LIN {X 0,Y 524.943,Z 315.664,A -85,B 0,C 180,E1 -4750.039,E2 -4750.039} C_VEL
LIN {X 0,Y 524.487,Z 334.734,A -85,B 0,C 180,E1 -4753.056,E2 -4753.056} C_VEL
LIN {X 0,Y 524.293,Z 346.228,A -85,B 0,C 180,E1 -4754.846,E2 -4754.846} C_VEL
LIN {X 0,Y 525.936,Z 357.339,A -85,B 0,C 180,E1 -4755.048,E2 -4755.048} C_VEL
LIN {X 0,Y 525.54,Z 454.207,A -85,B 0,C 180,E1 -4756.393,E2 -4756.393} C_VEL
LIN {X 0,Y 525.313,Z 467.512,A -85,B 0,C 180,E1 -4756.731,E2 -4756.731} C_VEL
LIN {X 0,Y 525.043,Z 480.819,A -85,B 0,C 180,E1 -4757.241,E2 -4757.241} C_VEL
LIN {X 0,Y 524.811,Z 492.313,A -85,B 0,C 180,E1 -4757.845,E2 -4757.845} C_VEL
LIN {X 0,Y 524.527,Z 503.595,A -85,B 0,C 180,E1 -4758.602,E2 -4758.602} C_VEL
LIN {X 0,Y 524.201,Z 514.045,A -85,B 0,C 180,E1 -4759.475,E2 -4759.475} C_VEL
LIN {X 0,Y 523.995,Z 522.59,A -85,B 0,C 180,E1 -4760.349,E2 -4760.349} C_VEL
LIN {X 0,Y 523.801,Z 530.474,A -85,B 0,C 180,E1 -4761.319,E2 -4761.319} C_VEL
LIN {X 0,Y 523.605,Z 538.173,A -85,B 0,C 180,E1 -4762.481,E2 -4762.481} C_VEL
LIN {X 0,Y 523.482,Z 545.27,A -85,B 0,C 180,E1 -4763.835,E2 -4763.835} C_VEL
LIN {X 0,Y 523.383,Z 549.99,A -85,B 0,C 180,E1 -4764.993,E2 -4764.993} C_VEL
LIN {X 0,Y 523.443,Z 553.599,A -85,B 0,C 180,E1 -4766.151,E2 -4766.151} C_VEL
LIN {X 0,Y 523.367,Z 555.458,A -85,B 0,C 180,E1 -4766.922,E2 -4766.922} C_VEL
LIN {X 0,Y 523.334,Z 556.852,A -85,B 0,C 180,E1 -4767.692,E2 -4767.692} C_VEL
LIN {X 0,Y 523.25,Z 558.452,A -85,B 0,C 180,E1 -4769.231,E2 -4769.231} C_VEL
LIN {X 0,Y 523.247,Z 558.668,A -85,B 0,C 180,E1 -4770.001,E2 -4770.001} C_VEL
LIN {X 0,Y 523.274,Z 557.844,A -85,B 0,C 180,E1 -4771.54,E2 -4771.54} C_VEL
LIN {X 0,Y 523.334,Z 556.851,A -85,B 0,C 180,E1 -4772.309,E2 -4772.309} C_VEL
LIN {X 0,Y 523.368,Z 555.456,A -85,B 0,C 180,E1 -4773.08,E2 -4773.08} C_VEL
LIN {X 0,Y 523.424,Z 552.521,A -85,B 0,C 180,E1 -4774.236,E2 -4774.236} C_VEL
LIN {X 0,Y 523.461,Z 548.548,A -85,B 0,C 180,E1 -4775.393,E2 -4775.393} C_VEL
LIN {X 0,Y 523.515,Z 542.453,A -85,B 0,C 180,E1 -4776.743,E2 -4776.743} C_VEL
LIN {X 0,Y 523.667,Z 535.757,A -85,B 0,C 180,E1 -4777.907,E2 -4777.907} C_VEL
LIN {X 0,Y 523.88,Z 527.47,A -85,B 0,C 180,E1 -4779.07,E2 -4779.07} C_VEL
LIN {X 0,Y 524.072,Z 518.975,A -85,B 0,C 180,E1 -4780.04,E2 -4780.04} C_VEL
LIN {X 0,Y 524.352,Z 508.478,A -85,B 0,C 180,E1 -4781.011,E2 -4781.011} C_VEL
LIN {X 0,Y 524.634,Z 498.216,A -85,B 0,C 180,E1 -4781.78,E2 -4781.78} C_VEL
LIN {X 0,Y 524.943,Z 486.709,A -85,B 0,C 180,E1 -4782.468,E2 -4782.468} C_VEL
LIN {X 0,Y 525.177,Z 475.02,A -85,B 0,C 180,E1 -4783.003,E2 -4783.003} C_VEL
LIN {X 0,Y 525.393,Z 461.551,A -85,B 0,C 180,E1 -4783.44,E2 -4783.44} C_VEL
LIN {X 0,Y 525.574,Z 448.203,A -85,B 0,C 180,E1 -4783.706,E2 -4783.706} C_VEL
LIN {X 0,Y 525.813,Z 355.915,A -85,B 0,C 180,E1 -4784.975,E2 -4784.975} C_VEL
LIN {X 0,Y 524.25,Z 345.993,A -85,B 0,C 180,E1 -4785.173,E2 -4785.173} C_VEL
LIN {X 0,Y 524.694,Z 325.97,A -85,B 0,C 180,E1 -4788.307,E2 -4788.307} C_VEL
LIN {X 0,Y 525.128,Z 306.537,A -85,B 0,C 180,E1 -4791.389,E2 -4791.389} C_VEL
LIN {X 0,Y 525.254,Z 297.571,A -85,B 0,C 180,E1 -4792.832,E2 -4792.832} C_VEL
LIN {X 0,Y 523.921,Z 290.224,A -85,B 0,C 180,E1 -4794.108,E2 -4794.108} C_VEL
LIN {X 0,Y 523.948,Z 290.22,A -85,B 0,C 180,E1 -4797.134,E2 -4797.134} C_VEL
LIN {X 0,Y 523.939,Z 290.226,A -85,B 0,C 180,E1 -4799.756,E2 -4799.756} C_VEL
LIN {X 0,Y 523.936,Z 290.22,A -85,B 0,C 180,E1 -4802.45,E2 -4802.45} C_VEL
LIN {X 0,Y 523.92,Z 290.22,A -85,B 0,C 180,E1 -4805.227,E2 -4805.227} C_VEL
LIN {X 0,Y 523.915,Z 290.227,A -85,B 0,C 180,E1 -4808.102,E2 -4808.102} C_VEL
LIN {X 0,Y 523.955,Z 290.213,A -85,B 0,C 180,E1 -4811.31,E2 -4811.31} C_VEL
LIN {X 0,Y 523.939,Z 290.22,A -85,B 0,C 180,E1 -4814.689,E2 -4814.689} C_VEL
LIN {X 0,Y 523.944,Z 290.217,A -85,B 0,C 180,E1 -4817.88,E2 -4817.88} C_VEL
LIN {X 0,Y 523.92,Z 290.221,A -85,B 0,C 180,E1 -4820.915,E2 -4820.915} C_VEL
LIN {X 0,Y 523.896,Z 290.22,A -85,B 0,C 180,E1 -4823.825,E2 -4823.825} C_VEL
LIN {X 0,Y 523.942,Z 290.222,A -85,B 0,C 180,E1 -4826.636,E2 -4826.636} C_VEL
LIN {X 0,Y 523.95,Z 290.217,A -85,B 0,C 180,E1 -4829.355,E2 -4829.355} C_VEL
LIN {X 0,Y 523.947,Z 290.214,A -85,B 0,C 180,E1 -4832.288,E2 -4832.288} C_VEL
LIN {X 0,Y 523.907,Z 290.224,A -85,B 0,C 180,E1 -4835.427,E2 -4835.427} C_VEL
LIN {X 0,Y 523.938,Z 290.216,A -85,B 0,C 180,E1 -4837.939,E2 -4837.939} C_VEL
LIN {X 0,Y 523.974,Z 290.21,A -85,B 0,C 180,E1 -4840.408,E2 -4840.408} C_VEL
LIN {X 0,Y 523.955,Z 290.214,A -85,B 0,C 180,E1 -4842.837,E2 -4842.837} C_VEL
LIN {X 0,Y 523.977,Z 290.215,A -85,B 0,C 180,E1 -4845.236,E2 -4845.236} C_VEL
LIN {X 0,Y 524.014,Z 290.205,A -85,B 0,C 180,E1 -4848.394,E2 -4848.394} C_VEL
LIN {X 0,Y 523.986,Z 290.213,A -85,B 0,C 180,E1 -4851.516,E2 -4851.516} C_VEL
LIN {X 0,Y 524.033,Z 290.212,A -85,B 0,C 180,E1 -4853.841,E2 -4853.841} C_VEL
LIN {X 0,Y 524.033,Z 290.201,A -85,B 0,C 180,E1 -4856.925,E2 -4856.925} C_VEL
LIN {X 0,Y 524.116,Z 290.2,A -85,B 0,C 180,E1 -4860,E2 -4860} C_VEL
LIN {X 0,Y 524.038,Z 290.202,A -85,B 0,C 180,E1 -4863.075,E2 -4863.075} C_VEL
LIN {X 0,Y 524.028,Z 290.209,A -85,B 0,C 180,E1 -4866.159,E2 -4866.159} C_VEL
LIN {X 0,Y 523.987,Z 290.207,A -85,B 0,C 180,E1 -4869.262,E2 -4869.262} C_VEL
LIN {X 0,Y 524.001,Z 290.208,A -85,B 0,C 180,E1 -4871.738,E2 -4871.738} C_VEL
LIN {X 0,Y 523.995,Z 290.212,A -85,B 0,C 180,E1 -4875.052,E2 -4875.052} C_VEL
LIN {X 0,Y 523.948,Z 290.212,A -85,B 0,C 180,E1 -4877.97,E2 -4877.97} C_VEL
LIN {X 0,Y 523.973,Z 290.214,A -85,B 0,C 180,E1 -4880.41,E2 -4880.41} C_VEL
LIN {X 0,Y 523.911,Z 290.226,A -85,B 0,C 180,E1 -4882.894,E2 -4882.894} C_VEL
LIN {X 0,Y 523.931,Z 290.219,A -85,B 0,C 180,E1 -4885.42,E2 -4885.42} C_VEL
LIN {X 0,Y 523.919,Z 290.216,A -85,B 0,C 180,E1 -4888.002,E2 -4888.002} C_VEL
LIN {X 0,Y 523.941,Z 290.218,A -85,B 0,C 180,E1 -4890.854,E2 -4890.854} C_VEL
LIN {X 0,Y 523.932,Z 290.219,A -85,B 0,C 180,E1 -4893.73,E2 -4893.73} C_VEL
LIN {X 0,Y 523.901,Z 290.22,A -85,B 0,C 180,E1 -4896.401,E2 -4896.401} C_VEL
LIN {X 0,Y 523.923,Z 290.22,A -85,B 0,C 180,E1 -4899.085,E2 -4899.085} C_VEL
LIN {X 0,Y 523.943,Z 290.219,A -85,B 0,C 180,E1 -4902.12,E2 -4902.12} C_VEL
LIN {X 0,Y 523.941,Z 290.218,A -85,B 0,C 180,E1 -4905.311,E2 -4905.311} C_VEL
LIN {X 0,Y 523.89,Z 290.223,A -85,B 0,C 180,E1 -4906.901,E2 -4906.901} C_VEL
LIN {X 0,Y 523.213,Z 290.312,A -85,B 0,C 180,E1 -4907.543,E2 -4907.543} C_VEL
LIN {X 0,Y 520.366,Z 290.672,A -85,B 0,C 180,E1 -4908.584,E2 -4908.584} C_VEL
LIN {X 0,Y 517.968,Z 290.974,A -85,B 0,C 180,E1 -4909.423,E2 -4909.423} C_VEL
LIN {X 0,Y 516.943,Z 291.098,A -85,B 0,C 180,E1 -4910.071,E2 -4910.071} C_VEL
LIN {X 0,Y 516.861,Z 291.105,A -85,B 0,C 180,E1 -4910.29,E2 -4910.29} C_VEL
LIN {X 0,Y 516.848,Z 291.102,A -85,B 0,C 180,E1 -4913.251,E2 -4913.251} C_VEL
LIN {X 0,Y 516.884,Z 291.102,A -85,B 0,C 180,E1 -4916.119,E2 -4916.119} C_VEL
LIN {X 0,Y 516.96,Z 291.244,A -85,B 0,C 180,E1 -4918.668,E2 -4918.668} C_VEL
LIN {X 0,Y 517.503,Z 296.303,A -85,B 0,C 180,E1 -4919.61,E2 -4919.61} C_VEL
LIN {X 0,Y 517.294,Z 312.213,A -85,B 0,C 180,E1 -4922.488,E2 -4922.488} C_VEL
LIN {X 0,Y 517.239,Z 318.815,A -85,B 0,C 180,E1 -4923.684,E2 -4923.684} C_VEL
LIN {X 0,Y 519.136,Z 329.983,A -85,B 0,C 180,E1 -4923.905,E2 -4923.905} C_VEL
LIN {X 0,Y 518.627,Z 426.694,A -85,B 0,C 180,E1 -4925.272,E2 -4925.272} C_VEL
LIN {X 0,Y 518.413,Z 439.775,A -85,B 0,C 180,E1 -4925.619,E2 -4925.619} C_VEL
LIN {X 0,Y 518.18,Z 451.968,A -85,B 0,C 180,E1 -4926.097,E2 -4926.097} C_VEL
LIN {X 0,Y 517.912,Z 463.726,A -85,B 0,C 180,E1 -4926.72,E2 -4926.72} C_VEL
LIN {X 0,Y 517.595,Z 475.325,A -85,B 0,C 180,E1 -4927.515,E2 -4927.515} C_VEL
LIN {X 0,Y 517.267,Z 485.379,A -85,B 0,C 180,E1 -4928.374,E2 -4928.374} C_VEL
LIN {X 0,Y 517.028,Z 494.258,A -85,B 0,C 180,E1 -4929.303,E2 -4929.303} C_VEL
LIN {X 0,Y 516.78,Z 502.321,A -85,B 0,C 180,E1 -4930.33,E2 -4930.33} C_VEL
LIN {X 0,Y 516.573,Z 510.116,A -85,B 0,C 180,E1 -4931.559,E2 -4931.559} C_VEL
LIN {X 0,Y 516.487,Z 515.377,A -85,B 0,C 180,E1 -4932.58,E2 -4932.58} C_VEL
LIN {X 0,Y 516.352,Z 520.412,A -85,B 0,C 180,E1 -4933.798,E2 -4933.798} C_VEL
LIN {X 0,Y 516.305,Z 524.542,A -85,B 0,C 180,E1 -4935.121,E2 -4935.121} C_VEL
LIN {X 0,Y 516.198,Z 527.693,A -85,B 0,C 180,E1 -4936.617,E2 -4936.617} C_VEL
LIN {X 0,Y 516.249,Z 529.366,A -85,B 0,C 180,E1 -4938.217,E2 -4938.217} C_VEL
LIN {X 0,Y 516.259,Z 529.606,A -85,B 0,C 180,E1 -4939.013,E2 -4939.013} C_VEL
LIN {X 0,Y 516.241,Z 529.405,A -85,B 0,C 180,E1 -4939.806,E2 -4939.806} C_VEL
LIN {X 0,Y 516.215,Z 527.808,A -85,B 0,C 180,E1 -4941.387,E2 -4941.387} C_VEL
LIN {X 0,Y 516.273,Z 526.41,A -85,B 0,C 180,E1 -4942.176,E2 -4942.176} C_VEL
LIN {X 0,Y 516.318,Z 522.893,A -85,B 0,C 180,E1 -4943.548,E2 -4943.548} C_VEL
LIN {X 0,Y 516.383,Z 517.948,A -85,B 0,C 180,E1 -4944.924,E2 -4944.924} C_VEL
LIN {X 0,Y 516.536,Z 512.457,A -85,B 0,C 180,E1 -4946.099,E2 -4946.099} C_VEL
LIN {X 0,Y 516.647,Z 505.638,A -85,B 0,C 180,E1 -4947.271,E2 -4947.271} C_VEL
LIN {X 0,Y 516.968,Z 497.099,A -85,B 0,C 180,E1 -4948.441,E2 -4948.441} C_VEL
LIN {X 0,Y 517.173,Z 488.4,A -85,B 0,C 180,E1 -4949.415,E2 -4949.415} C_VEL
LIN {X 0,Y 517.449,Z 477.72,A -85,B 0,C 180,E1 -4950.389,E2 -4950.389} C_VEL
LIN {X 0,Y 517.843,Z 466.961,A -85,B 0,C 180,E1 -4951.166,E2 -4951.166} C_VEL
LIN {X 0,Y 518.127,Z 454.986,A -85,B 0,C 180,E1 -4951.846,E2 -4951.846} C_VEL
LIN {X 0,Y 518.343,Z 442.502,A -85,B 0,C 180,E1 -4952.379,E2 -4952.379} C_VEL
LIN {X 0,Y 518.557,Z 430.182,A -85,B 0,C 180,E1 -4952.743,E2 -4952.743} C_VEL
LIN {X 0,Y 518.683,Z 414.633,A -85,B 0,C 180,E1 -4953.009,E2 -4953.009} C_VEL
LIN {X 0,Y 519.008,Z 328.91,A -85,B 0,C 180,E1 -4954.204,E2 -4954.204} C_VEL
LIN {X 0,Y 517.196,Z 318.905,A -85,B 0,C 180,E1 -4954.408,E2 -4954.408} C_VEL
LIN {X 0,Y 517.583,Z 301.777,A -85,B 0,C 180,E1 -4957.59,E2 -4957.59} C_VEL
LIN {X 0,Y 517.593,Z 295.417,A -85,B 0,C 180,E1 -4958.786,E2 -4958.786} C_VEL
LIN {X 0,Y 516.941,Z 291.096,A -85,B 0,C 180,E1 -4959.636,E2 -4959.636} C_VEL
LIN {X 0,Y 516.907,Z 291.095,A -85,B 0,C 180,E1 -4962.564,E2 -4962.564} C_VEL
LIN {X 0,Y 516.946,Z 291.086,A -85,B 0,C 180,E1 -4965.145,E2 -4965.145} C_VEL
LIN {X 0,Y 516.877,Z 291.101,A -85,B 0,C 180,E1 -4968.223,E2 -4968.223} C_VEL
LIN {X 0,Y 516.901,Z 291.093,A -85,B 0,C 180,E1 -4970.701,E2 -4970.701} C_VEL
LIN {X 0,Y 516.857,Z 291.097,A -85,B 0,C 180,E1 -4973.223,E2 -4973.223} C_VEL
LIN {X 0,Y 516.868,Z 291.104,A -85,B 0,C 180,E1 -4976.178,E2 -4976.178} C_VEL
LIN {X 0,Y 516.902,Z 291.091,A -85,B 0,C 180,E1 -4979.305,E2 -4979.305} C_VEL
LIN {X 0,Y 516.89,Z 291.102,A -85,B 0,C 180,E1 -4982.541,E2 -4982.541} C_VEL
LIN {X 0,Y 516.851,Z 291.098,A -85,B 0,C 180,E1 -4985.326,E2 -4985.326} C_VEL
LIN {X 0,Y 516.868,Z 291.106,A -85,B 0,C 180,E1 -4988.716,E2 -4988.716} C_VEL
LIN {X 0,Y 516.84,Z 291.099,A -85,B 0,C 180,E1 -4991.781,E2 -4991.781} C_VEL
LIN {X 0,Y 516.891,Z 291.101,A -85,B 0,C 180,E1 -4995.006,E2 -4995.006} C_VEL
LIN {X 0,Y 516.845,Z 291.1,A -85,B 0,C 180,E1 -4998.406,E2 -4998.406} C_VEL
LIN {X 0,Y 516.865,Z 291.103,A -85,B 0,C 180,E1 -5001.282,E2 -5001.282} C_VEL
LIN {X 0,Y 516.844,Z 291.101,A -85,B 0,C 180,E1 -5004.672,E2 -5004.672} C_VEL
LIN {X 0,Y 516.856,Z 291.104,A -85,B 0,C 180,E1 -5007.462,E2 -5007.462} C_VEL
LIN {X 0,Y 516.836,Z 291.1,A -85,B 0,C 180,E1 -5010.489,E2 -5010.489} C_VEL
LIN {X 0,Y 516.818,Z 291.109,A -85,B 0,C 180,E1 -5013.336,E2 -5013.336} C_VEL
LIN {X 0,Y 516.86,Z 291.101,A -85,B 0,C 180,E1 -5015.925,E2 -5015.925} C_VEL
LIN {X 0,Y 516.869,Z 291.096,A -85,B 0,C 180,E1 -5018.461,E2 -5018.461} C_VEL
LIN {X 0,Y 516.861,Z 291.097,A -85,B 0,C 180,E1 -5020.953,E2 -5020.953} C_VEL
LIN {X 0,Y 516.818,Z 291.106,A -85,B 0,C 180,E1 -5023.407,E2 -5023.407} C_VEL
LIN {X 0,Y 516.844,Z 291.108,A -85,B 0,C 180,E1 -5025.832,E2 -5025.832} C_VEL
LIN {X 0,Y 516.916,Z 291.095,A -85,B 0,C 180,E1 -5028.232,E2 -5028.232} C_VEL
LIN {X 0,Y 516.909,Z 291.092,A -85,B 0,C 180,E1 -5031.398,E2 -5031.398} C_VEL
LIN {X 0,Y 516.97,Z 291.087,A -85,B 0,C 180,E1 -5034.539,E2 -5034.539} C_VEL
LIN {X 0,Y 517.062,Z 291.073,A -85,B 0,C 180,E1 -5037.663,E2 -5037.663} C_VEL
LIN {X 0,Y 517.079,Z 291.073,A -85,B 0,C 180,E1 -5040.779,E2 -5040.779} C_VEL
LIN {X 0,Y 516.957,Z 291.085,A -85,B 0,C 180,E1 -5043.117,E2 -5043.117} C_VEL
LIN {X 0,Y 516.972,Z 291.088,A -85,B 0,C 180,E1 -5046.244,E2 -5046.244} C_VEL
LIN {X 0,Y 516.922,Z 291.089,A -85,B 0,C 180,E1 -5049.39,E2 -5049.39} C_VEL
LIN {X 0,Y 516.943,Z 291.086,A -85,B 0,C 180,E1 -5051.807,E2 -5051.807} C_VEL
LIN {X 0,Y 516.927,Z 291.093,A -85,B 0,C 180,E1 -5055.143,E2 -5055.143} C_VEL
LIN {X 0,Y 516.902,Z 291.092,A -85,B 0,C 180,E1 -5058.223,E2 -5058.223} C_VEL
LIN {X 0,Y 516.895,Z 291.097,A -85,B 0,C 180,E1 -5060.702,E2 -5060.702} C_VEL
LIN {X 0,Y 516.876,Z 291.095,A -85,B 0,C 180,E1 -5064.074,E2 -5064.074} C_VEL
LIN {X 0,Y 516.894,Z 291.095,A -85,B 0,C 180,E1 -5066.66,E2 -5066.66} C_VEL
LIN {X 0,Y 516.9,Z 291.097,A -85,B 0,C 180,E1 -5069.524,E2 -5069.524} C_VEL
LIN {X 0,Y 516.888,Z 291.093,A -85,B 0,C 180,E1 -5072.544,E2 -5072.544} C_VEL
LIN {X 0,Y 516.856,Z 291.105,A -85,B 0,C 180,E1 -5075.33,E2 -5075.33} C_VEL
LIN {X 0,Y 516.871,Z 291.099,A -85,B 0,C 180,E1 -5077.943,E2 -5077.943} C_VEL
LIN {X 0,Y 516.875,Z 291.095,A -85,B 0,C 180,E1 -5080.743,E2 -5080.743} C_VEL
LIN {X 0,Y 516.875,Z 291.102,A -85,B 0,C 180,E1 -5083.904,E2 -5083.904} C_VEL
LIN {X 0,Y 516.876,Z 291.1,A -85,B 0,C 180,E1 -5086.108,E2 -5086.108} C_VEL
LIN {X 0,Y 516.877,Z 291.096,A -85,B 0,C 180,E1 -5089.259,E2 -5089.259} C_VEL
LIN {X 0,Y 516.857,Z 291.102,A -85,B 0,C 180,E1 -5092.275,E2 -5092.275} C_VEL
LIN {X 0,Y 516.878,Z 291.094,A -85,B 0,C 180,E1 -5095.176,E2 -5095.176} C_VEL
LIN {X 0,Y 516.871,Z 291.102,A -85,B 0,C 180,E1 -5097.976,E2 -5097.976} C_VEL
LIN {X 0,Y 516.918,Z 291.094,A -85,B 0,C 180,E1 -5100.696,E2 -5100.696} C_VEL
LIN {X 0,Y 516.9,Z 291.096,A -85,B 0,C 180,E1 -5103.814,E2 -5103.814} C_VEL
LIN {X 0,Y 516.91,Z 291.275,A -85,B 0,C 180,E1 -5105.728,E2 -5105.728} C_VEL
LIN {X 0,Y 518.388,Z 299.806,A -85,B 0,C 180,E1 -5107.206,E2 -5107.206} C_VEL
LIN {X 0,Y 517.915,Z 318.019,A -85,B 0,C 180,E1 -5110.17,E2 -5110.17} C_VEL
LIN {X 0,Y 517.456,Z 335.805,A -85,B 0,C 180,E1 -5113.022,E2 -5113.022} C_VEL
LIN {X 0,Y 517.281,Z 346.006,A -85,B 0,C 180,E1 -5114.635,E2 -5114.635} C_VEL
LIN {X 0,Y 519.07,Z 358.553,A -85,B 0,C 180,E1 -5114.865,E2 -5114.865} C_VEL
LIN {X 0,Y 518.653,Z 453.984,A -85,B 0,C 180,E1 -5116.208,E2 -5116.208} C_VEL
LIN {X 0,Y 518.387,Z 467.297,A -85,B 0,C 180,E1 -5116.551,E2 -5116.551} C_VEL
LIN {X 0,Y 518.134,Z 480.61,A -85,B 0,C 180,E1 -5117.068,E2 -5117.068} C_VEL
LIN {X 0,Y 517.823,Z 493.124,A -85,B 0,C 180,E1 -5117.742,E2 -5117.742} C_VEL
LIN {X 0,Y 517.51,Z 504.686,A -85,B 0,C 180,E1 -5118.545,E2 -5118.545} C_VEL
LIN {X 0,Y 517.154,Z 514.888,A -85,B 0,C 180,E1 -5119.429,E2 -5119.429} C_VEL
LIN {X 0,Y 516.931,Z 524.07,A -85,B 0,C 180,E1 -5120.414,E2 -5120.414} C_VEL
LIN {X 0,Y 516.661,Z 533.013,A -85,B 0,C 180,E1 -5121.592,E2 -5121.592} C_VEL
LIN {X 0,Y 516.508,Z 540.213,A -85,B 0,C 180,E1 -5122.77,E2 -5122.77} C_VEL
LIN {X 0,Y 516.417,Z 546.769,A -85,B 0,C 180,E1 -5124.142,E2 -5124.142} C_VEL
LIN {X 0,Y 516.269,Z 551.103,A -85,B 0,C 180,E1 -5125.316,E2 -5125.316} C_VEL
LIN {X 0,Y 516.352,Z 553.401,A -85,B 0,C 180,E1 -5126.098,E2 -5126.098} C_VEL
LIN {X 0,Y 516.282,Z 555.26,A -85,B 0,C 180,E1 -5126.879,E2 -5126.879} C_VEL
LIN {X 0,Y 516.26,Z 556.654,A -85,B 0,C 180,E1 -5127.66,E2 -5127.66} C_VEL
LIN {X 0,Y 516.16,Z 558.254,A -85,B 0,C 180,E1 -5129.22,E2 -5129.22} C_VEL
LIN {X 0,Y 516.155,Z 558.469,A -85,B 0,C 180,E1 -5130.001,E2 -5130.001} C_VEL
LIN {X 0,Y 516.191,Z 557.646,A -85,B 0,C 180,E1 -5131.561,E2 -5131.561} C_VEL
LIN {X 0,Y 516.26,Z 556.652,A -85,B 0,C 180,E1 -5132.341,E2 -5132.341} C_VEL
LIN {X 0,Y 516.283,Z 555.256,A -85,B 0,C 180,E1 -5133.122,E2 -5133.122} C_VEL
LIN {X 0,Y 516.312,Z 552.32,A -85,B 0,C 180,E1 -5134.294,E2 -5134.294} C_VEL
LIN {X 0,Y 516.375,Z 548.346,A -85,B 0,C 180,E1 -5135.467,E2 -5135.467} C_VEL
LIN {X 0,Y 516.422,Z 543.132,A -85,B 0,C 180,E1 -5136.664,E2 -5136.664} C_VEL
LIN {X 0,Y 516.581,Z 536.79,A -85,B 0,C 180,E1 -5137.82,E2 -5137.82} C_VEL
LIN {X 0,Y 516.785,Z 528.756,A -85,B 0,C 180,E1 -5138.998,E2 -5138.998} C_VEL
LIN {X 0,Y 517.018,Z 520.569,A -85,B 0,C 180,E1 -5139.981,E2 -5139.981} C_VEL
LIN {X 0,Y 517.326,Z 510.586,A -85,B 0,C 180,E1 -5140.965,E2 -5140.965} C_VEL
LIN {X 0,Y 517.628,Z 500.738,A -85,B 0,C 180,E1 -5141.752,E2 -5141.752} C_VEL
LIN {X 0,Y 517.916,Z 489.603,A -85,B 0,C 180,E1 -5142.465,E2 -5142.465} C_VEL
LIN {X 0,Y 518.177,Z 477.153,A -85,B 0,C 180,E1 -5143.082,E2 -5143.082} C_VEL
LIN {X 0,Y 518.424,Z 464.071,A -85,B 0,C 180,E1 -5143.549,E2 -5143.549} C_VEL
LIN {X 0,Y 518.65,Z 451.001,A -85,B 0,C 180,E1 -5143.843,E2 -5143.843} C_VEL
LIN {X 0,Y 518.987,Z 356.904,A -85,B 0,C 180,E1 -5145.16,E2 -5145.16} C_VEL
LIN {X 0,Y 517.241,Z 345.723,A -85,B 0,C 180,E1 -5145.393,E2 -5145.393} C_VEL
LIN {X 0,Y 517.691,Z 326.778,A -85,B 0,C 180,E1 -5148.399,E2 -5148.399} C_VEL
LIN {X 0,Y 518.168,Z 307.605,A -85,B 0,C 180,E1 -5151.482,E2 -5151.482} C_VEL
LIN {X 0,Y 518.305,Z 298.878,A -85,B 0,C 180,E1 -5152.908,E2 -5152.908} C_VEL
LIN {X 0,Y 516.914,Z 291.097,A -85,B 0,C 180,E1 -5154.273,E2 -5154.273} C_VEL
LIN {X 0,Y 516.925,Z 291.1,A -85,B 0,C 180,E1 -5157.533,E2 -5157.533} C_VEL
LIN {X 0,Y 516.889,Z 291.102,A -85,B 0,C 180,E1 -5160.204,E2 -5160.204} C_VEL
LIN {X 0,Y 516.897,Z 291.095,A -85,B 0,C 180,E1 -5162.947,E2 -5162.947} C_VEL
LIN {X 0,Y 516.87,Z 291.104,A -85,B 0,C 180,E1 -5165.781,E2 -5165.781} C_VEL
LIN {X 0,Y 516.879,Z 291.097,A -85,B 0,C 180,E1 -5168.716,E2 -5168.716} C_VEL
LIN {X 0,Y 516.908,Z 291.094,A -85,B 0,C 180,E1 -5171.776,E2 -5171.776} C_VEL
LIN {X 0,Y 516.897,Z 291.094,A -85,B 0,C 180,E1 -5175.007,E2 -5175.007} C_VEL
LIN {X 0,Y 516.911,Z 291.1,A -85,B 0,C 180,E1 -5178.399,E2 -5178.399} C_VEL
LIN {X 0,Y 516.88,Z 291.094,A -85,B 0,C 180,E1 -5181.284,E2 -5181.284} C_VEL
LIN {X 0,Y 516.869,Z 291.098,A -85,B 0,C 180,E1 -5184.219,E2 -5184.219} C_VEL
LIN {X 0,Y 516.896,Z 291.097,A -85,B 0,C 180,E1 -5187.053,E2 -5187.053} C_VEL
LIN {X 0,Y 516.887,Z 291.094,A -85,B 0,C 180,E1 -5189.796,E2 -5189.796} C_VEL
LIN {X 0,Y 516.9,Z 291.093,A -85,B 0,C 180,E1 -5192.466,E2 -5192.466} C_VEL
LIN {X 0,Y 516.849,Z 291.106,A -85,B 0,C 180,E1 -5195.069,E2 -5195.069} C_VEL
LIN {X 0,Y 516.87,Z 291.099,A -85,B 0,C 180,E1 -5197.622,E2 -5197.622} C_VEL
LIN {X 0,Y 516.932,Z 291.088,A -85,B 0,C 180,E1 -5200.13,E2 -5200.13} C_VEL
LIN {X 0,Y 516.906,Z 291.09,A -85,B 0,C 180,E1 -5202.595,E2 -5202.595} C_VEL
LIN {X 0,Y 516.943,Z 291.088,A -85,B 0,C 180,E1 -5205.03,E2 -5205.03} C_VEL
LIN {X 0,Y 516.967,Z 291.084,A -85,B 0,C 180,E1 -5208.234,E2 -5208.234} C_VEL
LIN {X 0,Y 516.954,Z 291.088,A -85,B 0,C 180,E1 -5211.4,E2 -5211.4} C_VEL
LIN {X 0,Y 516.999,Z 291.086,A -85,B 0,C 180,E1 -5213.757,E2 -5213.757} C_VEL
LIN {X 0,Y 516.975,Z 291.08,A -85,B 0,C 180,E1 -5216.883,E2 -5216.883} C_VEL
LIN {X 0,Y 517.091,Z 291.067,A -85,B 0,C 180,E1 -5219.221,E2 -5219.221} C_VEL
LIN {X 0,Y 517.08,Z 291.076,A -85,B 0,C 180,E1 -5222.337,E2 -5222.337} C_VEL
LIN {X 0,Y 517.021,Z 291.074,A -85,B 0,C 180,E1 -5225.46,E2 -5225.46} C_VEL
LIN {X 0,Y 516.964,Z 291.088,A -85,B 0,C 180,E1 -5228.601,E2 -5228.601} C_VEL
LIN {X 0,Y 516.953,Z 291.086,A -85,B 0,C 180,E1 -5231.807,E2 -5231.807} C_VEL
LIN {X 0,Y 516.946,Z 291.089,A -85,B 0,C 180,E1 -5235.147,E2 -5235.147} C_VEL
LIN {X 0,Y 516.917,Z 291.089,A -85,B 0,C 180,E1 -5238.223,E2 -5238.223} C_VEL
LIN {X 0,Y 516.914,Z 291.097,A -85,B 0,C 180,E1 -5240.702,E2 -5240.702} C_VEL
LIN {X 0,Y 516.89,Z 291.092,A -85,B 0,C 180,E1 -5244.073,E2 -5244.073} C_VEL
LIN {X 0,Y 516.9,Z 291.094,A -85,B 0,C 180,E1 -5246.66,E2 -5246.66} C_VEL
LIN {X 0,Y 516.911,Z 291.095,A -85,B 0,C 180,E1 -5249.523,E2 -5249.523} C_VEL
LIN {X 0,Y 516.896,Z 291.092,A -85,B 0,C 180,E1 -5252.543,E2 -5252.543} C_VEL
LIN {X 0,Y 516.867,Z 291.103,A -85,B 0,C 180,E1 -5255.329,E2 -5255.329} C_VEL
LIN {X 0,Y 516.881,Z 291.099,A -85,B 0,C 180,E1 -5257.943,E2 -5257.943} C_VEL
LIN {X 0,Y 516.874,Z 291.096,A -85,B 0,C 180,E1 -5260.743,E2 -5260.743} C_VEL
LIN {X 0,Y 516.884,Z 291.102,A -85,B 0,C 180,E1 -5263.893,E2 -5263.893} C_VEL
LIN {X 0,Y 516.843,Z 291.101,A -85,B 0,C 180,E1 -5266.902,E2 -5266.902} C_VEL
LIN {X 0,Y 516.864,Z 291.102,A -85,B 0,C 180,E1 -5269.593,E2 -5269.593} C_VEL
LIN {X 0,Y 516.861,Z 291.105,A -85,B 0,C 180,E1 -5270.29,E2 -5270.29} C_VEL
LIN {X 0,Y 516.2,Z 291.183,A -85,B 0,C 180,E1 -5270.941,E2 -5270.941} C_VEL
LIN {X 0,Y 513.349,Z 291.543,A -85,B 0,C 180,E1 -5271.996,E2 -5271.996} C_VEL
LIN {X 0,Y 510.932,Z 291.844,A -85,B 0,C 180,E1 -5272.847,E2 -5272.847} C_VEL
LIN {X 0,Y 509.891,Z 291.971,A -85,B 0,C 180,E1 -5273.503,E2 -5273.503} C_VEL
LIN {X 0,Y 509.804,Z 291.982,A -85,B 0,C 180,E1 -5273.726,E2 -5273.726} C_VEL
LIN {X 0,Y 509.844,Z 291.98,A -85,B 0,C 180,E1 -5276.538,E2 -5276.538} C_VEL
LIN {X 0,Y 509.887,Z 292.074,A -85,B 0,C 180,E1 -5278.525,E2 -5278.525} C_VEL
LIN {X 0,Y 510.514,Z 297.753,A -85,B 0,C 180,E1 -5279.597,E2 -5279.597} C_VEL
LIN {X 0,Y 510.296,Z 313.783,A -85,B 0,C 180,E1 -5282.524,E2 -5282.524} C_VEL
LIN {X 0,Y 510.289,Z 319.229,A -85,B 0,C 180,E1 -5283.478,E2 -5283.478} C_VEL
LIN {X 0,Y 512.298,Z 331.341,A -85,B 0,C 180,E1 -5283.714,E2 -5283.714} C_VEL
LIN {X 0,Y 511.745,Z 426.106,A -85,B 0,C 180,E1 -5285.066,E2 -5285.066} C_VEL
LIN {X 0,Y 511.517,Z 439.542,A -85,B 0,C 180,E1 -5285.421,E2 -5285.421} C_VEL
LIN {X 0,Y 511.286,Z 452.079,A -85,B 0,C 180,E1 -5285.916,E2 -5285.916} C_VEL
LIN {X 0,Y 510.952,Z 464.688,A -85,B 0,C 180,E1 -5286.599,E2 -5286.599} C_VEL
LIN {X 0,Y 510.602,Z 476.585,A -85,B 0,C 180,E1 -5287.438,E2 -5287.438} C_VEL
LIN {X 0,Y 510.269,Z 487.146,A -85,B 0,C 180,E1 -5288.381,E2 -5288.381} C_VEL
LIN {X 0,Y 509.984,Z 495.942,A -85,B 0,C 180,E1 -5289.349,E2 -5289.349} C_VEL
LIN {X 0,Y 509.712,Z 504.253,A -85,B 0,C 180,E1 -5290.466,E2 -5290.466} C_VEL
LIN {X 0,Y 509.501,Z 511.63,A -85,B 0,C 180,E1 -5291.691,E2 -5291.691} C_VEL
LIN {X 0,Y 509.405,Z 516.726,A -85,B 0,C 180,E1 -5292.745,E2 -5292.745} C_VEL
LIN {X 0,Y 509.277,Z 521.514,A -85,B 0,C 180,E1 -5293.978,E2 -5293.978} C_VEL
LIN {X 0,Y 509.232,Z 524.662,A -85,B 0,C 180,E1 -5295.037,E2 -5295.037} C_VEL
LIN {X 0,Y 509.114,Z 527.642,A -85,B 0,C 180,E1 -5296.427,E2 -5296.427} C_VEL
LIN {X 0,Y 509.111,Z 528.773,A -85,B 0,C 180,E1 -5297.239,E2 -5297.239} C_VEL
LIN {X 0,Y 509.185,Z 529.706,A -85,B 0,C 180,E1 -5298.516,E2 -5298.516} C_VEL
LIN {X 0,Y 509.141,Z 529.685,A -85,B 0,C 180,E1 -5299.662,E2 -5299.662} C_VEL
LIN {X 0,Y 509.086,Z 529.156,A -85,B 0,C 180,E1 -5300.464,E2 -5300.464} C_VEL
LIN {X 0,Y 509.175,Z 526.895,A -85,B 0,C 180,E1 -5302.066,E2 -5302.066} C_VEL
LIN {X 0,Y 509.206,Z 525.153,A -85,B 0,C 180,E1 -5302.864,E2 -5302.864} C_VEL
LIN {X 0,Y 509.296,Z 521.684,A -85,B 0,C 180,E1 -5304.059,E2 -5304.059} C_VEL
LIN {X 0,Y 509.353,Z 517.141,A -85,B 0,C 180,E1 -5305.251,E2 -5305.251} C_VEL
LIN {X 0,Y 509.495,Z 510.276,A -85,B 0,C 180,E1 -5306.639,E2 -5306.639} C_VEL
LIN {X 0,Y 509.718,Z 502.866,A -85,B 0,C 180,E1 -5307.826,E2 -5307.826} C_VEL
LIN {X 0,Y 510.008,Z 495.313,A -85,B 0,C 180,E1 -5308.815,E2 -5308.815} C_VEL
LIN {X 0,Y 510.198,Z 486.217,A -85,B 0,C 180,E1 -5309.802,E2 -5309.802} C_VEL
LIN {X 0,Y 510.545,Z 476.089,A -85,B 0,C 180,E1 -5310.69,E2 -5310.69} C_VEL
LIN {X 0,Y 510.956,Z 464.871,A -85,B 0,C 180,E1 -5311.477,E2 -5311.477} C_VEL
LIN {X 0,Y 511.256,Z 453.283,A -85,B 0,C 180,E1 -5312.117,E2 -5312.117} C_VEL
LIN {X 0,Y 511.466,Z 440.646,A -85,B 0,C 180,E1 -5312.633,E2 -5312.633} C_VEL
LIN {X 0,Y 511.686,Z 427.164,A -85,B 0,C 180,E1 -5313.001,E2 -5313.001} C_VEL
LIN {X 0,Y 512.013,Z 378.332,A -85,B 0,C 180,E1 -5313.713,E2 -5313.713} C_VEL
LIN {X 0,Y 512.17,Z 329.763,A -85,B 0,C 180,E1 -5314.402,E2 -5314.402} C_VEL
LIN {X 0,Y 510.14,Z 318.975,A -85,B 0,C 180,E1 -5314.642,E2 -5314.642} C_VEL
LIN {X 0,Y 510.614,Z 302.684,A -85,B 0,C 180,E1 -5317.691,E2 -5317.691} C_VEL
LIN {X 0,Y 510.569,Z 296.28,A -85,B 0,C 180,E1 -5318.908,E2 -5318.908} C_VEL
LIN {X 0,Y 509.885,Z 291.975,A -85,B 0,C 180,E1 -5319.77,E2 -5319.77} C_VEL
LIN {X 0,Y 509.908,Z 291.972,A -85,B 0,C 180,E1 -5321.931,E2 -5321.931} C_VEL
LIN {X 0,Y 509.898,Z 291.965,A -85,B 0,C 180,E1 -5325.241,E2 -5325.241} C_VEL
LIN {X 0,Y 509.836,Z 291.975,A -85,B 0,C 180,E1 -5328.484,E2 -5328.484} C_VEL
LIN {X 0,Y 509.844,Z 291.971,A -85,B 0,C 180,E1 -5331.001,E2 -5331.001} C_VEL
LIN {X 0,Y 509.819,Z 291.975,A -85,B 0,C 180,E1 -5333.563,E2 -5333.563} C_VEL
LIN {X 0,Y 509.806,Z 291.984,A -85,B 0,C 180,E1 -5336.353,E2 -5336.353} C_VEL
LIN {X 0,Y 509.832,Z 291.975,A -85,B 0,C 180,E1 -5338.846,E2 -5338.846} C_VEL
LIN {X 0,Y 509.809,Z 291.975,A -85,B 0,C 180,E1 -5341.59,E2 -5341.59} C_VEL
LIN {X 0,Y 509.831,Z 291.98,A -85,B 0,C 180,E1 -5344.414,E2 -5344.414} C_VEL
LIN {X 0,Y 509.789,Z 291.978,A -85,B 0,C 180,E1 -5347.342,E2 -5347.342} C_VEL
LIN {X 0,Y 509.809,Z 291.979,A -85,B 0,C 180,E1 -5350.384,E2 -5350.384} C_VEL
LIN {X 0,Y 509.788,Z 291.978,A -85,B 0,C 180,E1 -5353.574,E2 -5353.574} C_VEL
LIN {X 0,Y 509.787,Z 291.98,A -85,B 0,C 180,E1 -5356.424,E2 -5356.424} C_VEL
LIN {X 0,Y 509.807,Z 291.977,A -85,B 0,C 180,E1 -5359.614,E2 -5359.614} C_VEL
LIN {X 0,Y 509.776,Z 291.982,A -85,B 0,C 180,E1 -5362.655,E2 -5362.655} C_VEL
LIN {X 0,Y 509.825,Z 291.975,A -85,B 0,C 180,E1 -5365.801,E2 -5365.801} C_VEL
LIN {X 0,Y 509.806,Z 291.977,A -85,B 0,C 180,E1 -5368.725,E2 -5368.725} C_VEL
LIN {X 0,Y 509.815,Z 291.976,A -85,B 0,C 180,E1 -5372.049,E2 -5372.049} C_VEL
LIN {X 0,Y 509.775,Z 291.979,A -85,B 0,C 180,E1 -5374.698,E2 -5374.698} C_VEL
LIN {X 0,Y 509.817,Z 291.981,A -85,B 0,C 180,E1 -5377.458,E2 -5377.458} C_VEL
LIN {X 0,Y 509.895,Z 291.972,A -85,B 0,C 180,E1 -5379.844,E2 -5379.844} C_VEL
LIN {X 0,Y 509.773,Z 291.981,A -85,B 0,C 180,E1 -5383.171,E2 -5383.171} C_VEL
LIN {X 0,Y 509.807,Z 291.981,A -85,B 0,C 180,E1 -5385.632,E2 -5385.632} C_VEL
LIN {X 0,Y 509.88,Z 291.973,A -85,B 0,C 180,E1 -5388.13,E2 -5388.13} C_VEL
LIN {X 0,Y 509.862,Z 291.969,A -85,B 0,C 180,E1 -5391.279,E2 -5391.279} C_VEL
LIN {X 0,Y 509.906,Z 291.966,A -85,B 0,C 180,E1 -5393.669,E2 -5393.669} C_VEL
LIN {X 0,Y 509.906,Z 291.964,A -85,B 0,C 180,E1 -5396.839,E2 -5396.839} C_VEL
LIN {X 0,Y 509.918,Z 291.969,A -85,B 0,C 180,E1 -5398.42,E2 -5398.42} C_VEL
LIN {X 0,Y 510.028,Z 291.951,A -85,B 0,C 180,E1 -5400.789,E2 -5400.789} C_VEL
LIN {X 0,Y 509.899,Z 291.964,A -85,B 0,C 180,E1 -5403.16,E2 -5403.16} C_VEL
LIN {X 0,Y 509.926,Z 291.967,A -85,B 0,C 180,E1 -5406.33,E2 -5406.33} C_VEL
LIN {X 0,Y 509.872,Z 291.975,A -85,B 0,C 180,E1 -5408.721,E2 -5408.721} C_VEL
LIN {X 0,Y 509.895,Z 291.965,A -85,B 0,C 180,E1 -5411.932,E2 -5411.932} C_VEL
LIN {X 0,Y 509.885,Z 291.969,A -85,B 0,C 180,E1 -5415.242,E2 -5415.242} C_VEL
LIN {X 0,Y 509.847,Z 291.973,A -85,B 0,C 180,E1 -5418.484,E2 -5418.484} C_VEL
LIN {X 0,Y 509.837,Z 291.982,A -85,B 0,C 180,E1 -5421.002,E2 -5421.002} C_VEL
LIN {X 0,Y 509.809,Z 291.978,A -85,B 0,C 180,E1 -5423.564,E2 -5423.564} C_VEL
LIN {X 0,Y 509.863,Z 291.976,A -85,B 0,C 180,E1 -5427.057,E2 -5427.057} C_VEL
LIN {X 0,Y 509.849,Z 291.973,A -85,B 0,C 180,E1 -5429.752,E2 -5429.752} C_VEL
LIN {X 0,Y 509.865,Z 291.969,A -85,B 0,C 180,E1 -5432.775,E2 -5432.775} C_VEL
LIN {X 0,Y 509.816,Z 291.982,A -85,B 0,C 180,E1 -5435.579,E2 -5435.579} C_VEL
LIN {X 0,Y 509.842,Z 291.971,A -85,B 0,C 180,E1 -5438.339,E2 -5438.339} C_VEL
LIN {X 0,Y 509.846,Z 291.976,A -85,B 0,C 180,E1 -5441.427,E2 -5441.427} C_VEL
LIN {X 0,Y 509.833,Z 291.972,A -85,B 0,C 180,E1 -5444.671,E2 -5444.671} C_VEL
LIN {X 0,Y 509.845,Z 291.976,A -85,B 0,C 180,E1 -5448.105,E2 -5448.105} C_VEL
LIN {X 0,Y 509.841,Z 291.972,A -85,B 0,C 180,E1 -5450.648,E2 -5450.648} C_VEL
LIN {X 0,Y 509.805,Z 291.979,A -85,B 0,C 180,E1 -5453.646,E2 -5453.646} C_VEL
LIN {X 0,Y 509.856,Z 291.973,A -85,B 0,C 180,E1 -5456.54,E2 -5456.54} C_VEL
LIN {X 0,Y 509.84,Z 291.971,A -85,B 0,C 180,E1 -5459.335,E2 -5459.335} C_VEL
LIN {X 0,Y 509.881,Z 291.972,A -85,B 0,C 180,E1 -5462.055,E2 -5462.055} C_VEL
LIN {X 0,Y 509.811,Z 291.983,A -85,B 0,C 180,E1 -5464.701,E2 -5464.701} C_VEL
LIN {X 0,Y 509.853,Z 292.015,A -85,B 0,C 180,E1 -5465.54,E2 -5465.54} C_VEL
LIN {X 0,Y 511.45,Z 301.158,A -85,B 0,C 180,E1 -5467.144,E2 -5467.144} C_VEL
LIN {X 0,Y 510.97,Z 317.822,A -85,B 0,C 180,E1 -5469.889,E2 -5469.889} C_VEL
LIN {X 0,Y 510.505,Z 335.613,A -85,B 0,C 180,E1 -5472.784,E2 -5472.784} C_VEL
LIN {X 0,Y 510.268,Z 345.801,A -85,B 0,C 180,E1 -5474.419,E2 -5474.419} C_VEL
LIN {X 0,Y 512.234,Z 359.103,A -85,B 0,C 180,E1 -5474.669,E2 -5474.669} C_VEL
LIN {X 0,Y 511.76,Z 453.76,A -85,B 0,C 180,E1 -5476.019,E2 -5476.019} C_VEL
LIN {X 0,Y 511.485,Z 467.082,A -85,B 0,C 180,E1 -5476.366,E2 -5476.366} C_VEL
LIN {X 0,Y 511.179,Z 480.399,A -85,B 0,C 180,E1 -5476.889,E2 -5476.889} C_VEL
LIN {X 0,Y 510.903,Z 491.844,A -85,B 0,C 180,E1 -5477.505,E2 -5477.505} C_VEL
LIN {X 0,Y 510.563,Z 503.186,A -85,B 0,C 180,E1 -5478.286,E2 -5478.286} C_VEL
LIN {X 0,Y 510.212,Z 513.639,A -85,B 0,C 180,E1 -5479.183,E2 -5479.183} C_VEL
LIN {X 0,Y 509.94,Z 522.186,A -85,B 0,C 180,E1 -5480.081,E2 -5480.081} C_VEL
LIN {X 0,Y 509.681,Z 530.072,A -85,B 0,C 180,E1 -5481.077,E2 -5481.077} C_VEL
LIN {X 0,Y 509.479,Z 537.773,A -85,B 0,C 180,E1 -5482.271,E2 -5482.271} C_VEL
LIN {X 0,Y 509.319,Z 544.003,A -85,B 0,C 180,E1 -5483.473,E2 -5483.473} C_VEL
LIN {X 0,Y 509.243,Z 549.594,A -85,B 0,C 180,E1 -5484.854,E2 -5484.854} C_VEL
LIN {X 0,Y 509.245,Z 553.202,A -85,B 0,C 180,E1 -5486.044,E2 -5486.044} C_VEL
LIN {X 0,Y 509.2,Z 555.062,A -85,B 0,C 180,E1 -5486.836,E2 -5486.836} C_VEL
LIN {X 0,Y 509.189,Z 556.457,A -85,B 0,C 180,E1 -5487.627,E2 -5487.627} C_VEL
LIN {X 0,Y 509.073,Z 558.056,A -85,B 0,C 180,E1 -5489.21,E2 -5489.21} C_VEL
LIN {X 0,Y 509.066,Z 558.271,A -85,B 0,C 180,E1 -5490.001,E2 -5490.001} C_VEL
LIN {X 0,Y 509.112,Z 557.447,A -85,B 0,C 180,E1 -5491.583,E2 -5491.583} C_VEL
LIN {X 0,Y 509.189,Z 556.453,A -85,B 0,C 180,E1 -5492.374,E2 -5492.374} C_VEL
LIN {X 0,Y 509.201,Z 555.056,A -85,B 0,C 180,E1 -5493.165,E2 -5493.165} C_VEL
LIN {X 0,Y 509.204,Z 552.118,A -85,B 0,C 180,E1 -5494.354,E2 -5494.354} C_VEL
LIN {X 0,Y 509.293,Z 548.143,A -85,B 0,C 180,E1 -5495.544,E2 -5495.544} C_VEL
LIN {X 0,Y 509.4,Z 542.13,A -85,B 0,C 180,E1 -5496.914,E2 -5496.914} C_VEL
LIN {X 0,Y 509.545,Z 535.347,A -85,B 0,C 180,E1 -5498.128,E2 -5498.128} C_VEL
LIN {X 0,Y 509.782,Z 527.057,A -85,B 0,C 180,E1 -5499.323,E2 -5499.323} C_VEL
LIN {X 0,Y 510.015,Z 518.557,A -85,B 0,C 180,E1 -5500.32,E2 -5500.32} C_VEL
LIN {X 0,Y 510.394,Z 508.058,A -85,B 0,C 180,E1 -5501.316,E2 -5501.316} C_VEL
LIN {X 0,Y 510.687,Z 497.785,A -85,B 0,C 180,E1 -5502.107,E2 -5502.107} C_VEL
LIN {X 0,Y 511.05,Z 486.279,A -85,B 0,C 180,E1 -5502.812,E2 -5502.812} C_VEL
LIN {X 0,Y 511.358,Z 474.581,A -85,B 0,C 180,E1 -5503.36,E2 -5503.36} C_VEL
LIN {X 0,Y 511.576,Z 462.013,A -85,B 0,C 180,E1 -5503.785,E2 -5503.785} C_VEL
LIN {X 0,Y 511.788,Z 449.256,A -85,B 0,C 180,E1 -5504.058,E2 -5504.058} C_VEL
LIN {X 0,Y 512.168,Z 357.888,A -85,B 0,C 180,E1 -5505.35,E2 -5505.35} C_VEL
LIN {X 0,Y 510.234,Z 345.635,A -85,B 0,C 180,E1 -5505.591,E2 -5505.591} C_VEL
LIN {X 0,Y 510.692,Z 327.84,A -85,B 0,C 180,E1 -5508.453,E2 -5508.453} C_VEL
LIN {X 0,Y 511.217,Z 308.699,A -85,B 0,C 180,E1 -5511.577,E2 -5511.577} C_VEL
LIN {X 0,Y 511.394,Z 300.354,A -85,B 0,C 180,E1 -5512.961,E2 -5512.961} C_VEL
LIN {X 0,Y 509.84,Z 291.977,A -85,B 0,C 180,E1 -5514.484,E2 -5514.484} C_VEL
LIN {X 0,Y 509.876,Z 291.973,A -85,B 0,C 180,E1 -5517.056,E2 -5517.056} C_VEL
LIN {X 0,Y 509.859,Z 291.979,A -85,B 0,C 180,E1 -5519.751,E2 -5519.751} C_VEL
LIN {X 0,Y 509.876,Z 291.97,A -85,B 0,C 180,E1 -5522.774,E2 -5522.774} C_VEL
LIN {X 0,Y 509.825,Z 291.979,A -85,B 0,C 180,E1 -5525.578,E2 -5525.578} C_VEL
LIN {X 0,Y 509.85,Z 291.977,A -85,B 0,C 180,E1 -5528.338,E2 -5528.338} C_VEL
LIN {X 0,Y 509.854,Z 291.97,A -85,B 0,C 180,E1 -5531.426,E2 -5531.426} C_VEL
LIN {X 0,Y 509.84,Z 291.977,A -85,B 0,C 180,E1 -5534.67,E2 -5534.67} C_VEL
LIN {X 0,Y 509.851,Z 291.975,A -85,B 0,C 180,E1 -5538.104,E2 -5538.104} C_VEL
LIN {X 0,Y 509.846,Z 291.978,A -85,B 0,C 180,E1 -5540.647,E2 -5540.647} C_VEL
LIN {X 0,Y 509.81,Z 291.975,A -85,B 0,C 180,E1 -5543.646,E2 -5543.646} C_VEL
LIN {X 0,Y 509.86,Z 291.974,A -85,B 0,C 180,E1 -5546.539,E2 -5546.539} C_VEL
LIN {X 0,Y 509.843,Z 291.975,A -85,B 0,C 180,E1 -5549.334,E2 -5549.334} C_VEL
LIN {X 0,Y 509.851,Z 291.969,A -85,B 0,C 180,E1 -5552.052,E2 -5552.052} C_VEL
LIN {X 0,Y 509.807,Z 291.979,A -85,B 0,C 180,E1 -5554.7,E2 -5554.7} C_VEL
LIN {X 0,Y 509.826,Z 291.979,A -85,B 0,C 180,E1 -5557.458,E2 -5557.458} C_VEL
LIN {X 0,Y 509.917,Z 291.963,A -85,B 0,C 180,E1 -5559.845,E2 -5559.845} C_VEL
LIN {X 0,Y 509.873,Z 291.972,A -85,B 0,C 180,E1 -5563.174,E2 -5563.174} C_VEL
LIN {X 0,Y 509.861,Z 291.976,A -85,B 0,C 180,E1 -5565.634,E2 -5565.634} C_VEL
LIN {X 0,Y 509.912,Z 291.961,A -85,B 0,C 180,E1 -5568.875,E2 -5568.875} C_VEL
LIN {X 0,Y 509.921,Z 291.964,A -85,B 0,C 180,E1 -5572.078,E2 -5572.078} C_VEL
LIN {X 0,Y 509.975,Z 291.954,A -85,B 0,C 180,E1 -5574.464,E2 -5574.464} C_VEL
LIN {X 0,Y 510.05,Z 291.947,A -85,B 0,C 180,E1 -5577.631,E2 -5577.631} C_VEL
LIN {X 0,Y 510.058,Z 291.95,A -85,B 0,C 180,E1 -5580,E2 -5580} C_VEL
LIN {X 0,Y 510.05,Z 291.951,A -85,B 0,C 180,E1 -5582.369,E2 -5582.369} C_VEL
LIN {X 0,Y 509.972,Z 291.953,A -85,B 0,C 180,E1 -5585.536,E2 -5585.536} C_VEL
LIN {X 0,Y 509.91,Z 291.965,A -85,B 0,C 180,E1 -5588.72,E2 -5588.72} C_VEL
LIN {X 0,Y 509.906,Z 291.965,A -85,B 0,C 180,E1 -5591.932,E2 -5591.932} C_VEL
LIN {X 0,Y 509.896,Z 291.967,A -85,B 0,C 180,E1 -5595.242,E2 -5595.242} C_VEL
LIN {X 0,Y 509.862,Z 291.971,A -85,B 0,C 180,E1 -5598.484,E2 -5598.484} C_VEL
LIN {X 0,Y 509.852,Z 291.975,A -85,B 0,C 180,E1 -5601.002,E2 -5601.002} C_VEL
LIN {X 0,Y 509.822,Z 291.975,A -85,B 0,C 180,E1 -5603.564,E2 -5603.564} C_VEL
LIN {X 0,Y 509.881,Z 291.966,A -85,B 0,C 180,E1 -5606.371,E2 -5606.371} C_VEL
LIN {X 0,Y 509.86,Z 291.971,A -85,B 0,C 180,E1 -5609.726,E2 -5609.726} C_VEL
LIN {X 0,Y 509.869,Z 291.969,A -85,B 0,C 180,E1 -5612.773,E2 -5612.773} C_VEL
LIN {X 0,Y 509.826,Z 291.981,A -85,B 0,C 180,E1 -5615.578,E2 -5615.578} C_VEL
LIN {X 0,Y 509.852,Z 291.971,A -85,B 0,C 180,E1 -5618.338,E2 -5618.338} C_VEL
LIN {X 0,Y 509.848,Z 291.977,A -85,B 0,C 180,E1 -5621.427,E2 -5621.427} C_VEL
LIN {X 0,Y 509.842,Z 291.972,A -85,B 0,C 180,E1 -5624.67,E2 -5624.67} C_VEL
LIN {X 0,Y 509.806,Z 291.981,A -85,B 0,C 180,E1 -5627.507,E2 -5627.507} C_VEL
LIN {X 0,Y 509.836,Z 291.977,A -85,B 0,C 180,E1 -5630.646,E2 -5630.646} C_VEL
LIN {X 0,Y 509.804,Z 291.982,A -85,B 0,C 180,E1 -5633.726,E2 -5633.726} C_VEL
LIN {X 0,Y 509.139,Z 292.067,A -85,B 0,C 180,E1 -5634.386,E2 -5634.386} C_VEL
LIN {X 0,Y 506.31,Z 292.416,A -85,B 0,C 180,E1 -5635.458,E2 -5635.458} C_VEL
LIN {X 0,Y 503.917,Z 292.719,A -85,B 0,C 180,E1 -5636.321,E2 -5636.321} C_VEL
LIN {X 0,Y 502.884,Z 292.844,A -85,B 0,C 180,E1 -5636.988,E2 -5636.988} C_VEL
LIN {X 0,Y 502.796,Z 292.854,A -85,B 0,C 180,E1 -5637.213,E2 -5637.213} C_VEL
LIN {X 0,Y 502.846,Z 292.886,A -85,B 0,C 180,E1 -5638.365,E2 -5638.365} C_VEL
LIN {X 0,Y 503.547,Z 298.129,A -85,B 0,C 180,E1 -5639.374,E2 -5639.374} C_VEL
LIN {X 0,Y 503.338,Z 312.955,A -85,B 0,C 180,E1 -5642.111,E2 -5642.111} C_VEL
LIN {X 0,Y 503.289,Z 319.282,A -85,B 0,C 180,E1 -5643.251,E2 -5643.251} C_VEL
LIN {X 0,Y 505.47,Z 332.061,A -85,B 0,C 180,E1 -5643.509,E2 -5643.509} C_VEL
LIN {X 0,Y 504.86,Z 427.112,A -85,B 0,C 180,E1 -5644.891,E2 -5644.891} C_VEL
LIN {X 0,Y 504.621,Z 440.304,A -85,B 0,C 180,E1 -5645.251,E2 -5645.251} C_VEL
LIN {X 0,Y 504.385,Z 452.185,A -85,B 0,C 180,E1 -5645.729,E2 -5645.729} C_VEL
LIN {X 0,Y 504.074,Z 463.996,A -85,B 0,C 180,E1 -5646.369,E2 -5646.369} C_VEL
LIN {X 0,Y 503.684,Z 476.094,A -85,B 0,C 180,E1 -5647.222,E2 -5647.222} C_VEL
LIN {X 0,Y 503.274,Z 486.783,A -85,B 0,C 180,E1 -5648.173,E2 -5648.173} C_VEL
LIN {X 0,Y 502.997,Z 495.429,A -85,B 0,C 180,E1 -5649.124,E2 -5649.124} C_VEL
LIN {X 0,Y 502.715,Z 503.367,A -85,B 0,C 180,E1 -5650.183,E2 -5650.183} C_VEL
LIN {X 0,Y 502.456,Z 511.161,A -85,B 0,C 180,E1 -5651.466,E2 -5651.466} C_VEL
LIN {X 0,Y 502.346,Z 516.206,A -85,B 0,C 180,E1 -5652.494,E2 -5652.494} C_VEL
LIN {X 0,Y 502.195,Z 521.149,A -85,B 0,C 180,E1 -5653.746,E2 -5653.746} C_VEL
LIN {X 0,Y 502.143,Z 524.801,A -85,B 0,C 180,E1 -5654.957,E2 -5654.957} C_VEL
LIN {X 0,Y 502.045,Z 527.557,A -85,B 0,C 180,E1 -5656.232,E2 -5656.232} C_VEL
LIN {X 0,Y 502.011,Z 528.795,A -85,B 0,C 180,E1 -5657.056,E2 -5657.056} C_VEL
LIN {X 0,Y 502.103,Z 529.896,A -85,B 0,C 180,E1 -5658.466,E2 -5658.466} C_VEL
LIN {X 0,Y 502.046,Z 529.917,A -85,B 0,C 180,E1 -5659.514,E2 -5659.514} C_VEL
LIN {X 0,Y 502.005,Z 529.499,A -85,B 0,C 180,E1 -5660.328,E2 -5660.328} C_VEL
LIN {X 0,Y 502.04,Z 528.637,A -85,B 0,C 180,E1 -5661.141,E2 -5661.141} C_VEL
LIN {X 0,Y 502.095,Z 527.371,A -85,B 0,C 180,E1 -5661.953,E2 -5661.953} C_VEL
LIN {X 0,Y 502.138,Z 524.695,A -85,B 0,C 180,E1 -5663.167,E2 -5663.167} C_VEL
LIN {X 0,Y 502.253,Z 521.01,A -85,B 0,C 180,E1 -5664.378,E2 -5664.378} C_VEL
LIN {X 0,Y 502.332,Z 516.229,A -85,B 0,C 180,E1 -5665.586,E2 -5665.586} C_VEL
LIN {X 0,Y 502.439,Z 510.216,A -85,B 0,C 180,E1 -5666.792,E2 -5666.792} C_VEL
LIN {X 0,Y 502.698,Z 502.749,A -85,B 0,C 180,E1 -5667.996,E2 -5667.996} C_VEL
LIN {X 0,Y 503.033,Z 495.129,A -85,B 0,C 180,E1 -5668.999,E2 -5668.999} C_VEL
LIN {X 0,Y 503.268,Z 484.868,A -85,B 0,C 180,E1 -5670.099,E2 -5670.099} C_VEL
LIN {X 0,Y 503.672,Z 474.407,A -85,B 0,C 180,E1 -5670.999,E2 -5670.999} C_VEL
LIN {X 0,Y 504.102,Z 462.723,A -85,B 0,C 180,E1 -5671.797,E2 -5671.797} C_VEL
LIN {X 0,Y 504.427,Z 450.281,A -85,B 0,C 180,E1 -5672.445,E2 -5672.445} C_VEL
LIN {X 0,Y 504.668,Z 437.902,A -85,B 0,C 180,E1 -5672.918,E2 -5672.918} C_VEL
LIN {X 0,Y 504.847,Z 425.065,A -85,B 0,C 180,E1 -5673.241,E2 -5673.241} C_VEL
LIN {X 0,Y 505.389,Z 330.884,A -85,B 0,C 180,E1 -5674.599,E2 -5674.599} C_VEL
LIN {X 0,Y 503.128,Z 319.17,A -85,B 0,C 180,E1 -5674.857,E2 -5674.857} C_VEL
LIN {X 0,Y 503.591,Z 305.375,A -85,B 0,C 180,E1 -5677.457,E2 -5677.457} C_VEL
LIN {X 0,Y 503.688,Z 298.182,A -85,B 0,C 180,E1 -5678.828,E2 -5678.828} C_VEL
LIN {X 0,Y 502.861,Z 292.85,A -85,B 0,C 180,E1 -5679.908,E2 -5679.908} C_VEL
LIN {X 0,Y 502.848,Z 292.852,A -85,B 0,C 180,E1 -5682.101,E2 -5682.101} C_VEL
LIN {X 0,Y 502.848,Z 292.844,A -85,B 0,C 180,E1 -5685.399,E2 -5685.399} C_VEL
LIN {X 0,Y 502.809,Z 292.848,A -85,B 0,C 180,E1 -5688.752,E2 -5688.752} C_VEL
LIN {X 0,Y 502.78,Z 292.851,A -85,B 0,C 180,E1 -5691.31,E2 -5691.31} C_VEL
LIN {X 0,Y 502.767,Z 292.857,A -85,B 0,C 180,E1 -5693.914,E2 -5693.914} C_VEL
LIN {X 0,Y 502.781,Z 292.856,A -85,B 0,C 180,E1 -5696.57,E2 -5696.57} C_VEL
LIN {X 0,Y 502.792,Z 292.852,A -85,B 0,C 180,E1 -5699.929,E2 -5699.929} C_VEL
LIN {X 0,Y 502.8,Z 292.85,A -85,B 0,C 180,E1 -5703.033,E2 -5703.033} C_VEL
LIN {X 0,Y 502.758,Z 292.854,A -85,B 0,C 180,E1 -5705.951,E2 -5705.951} C_VEL
LIN {X 0,Y 502.778,Z 292.856,A -85,B 0,C 180,E1 -5708.977,E2 -5708.977} C_VEL
LIN {X 0,Y 502.741,Z 292.857,A -85,B 0,C 180,E1 -5712.191,E2 -5712.191} C_VEL
LIN {X 0,Y 502.773,Z 292.853,A -85,B 0,C 180,E1 -5715.47,E2 -5715.47} C_VEL
LIN {X 0,Y 502.757,Z 292.862,A -85,B 0,C 180,E1 -5718.927,E2 -5718.927} C_VEL
LIN {X 0,Y 502.754,Z 292.854,A -85,B 0,C 180,E1 -5722.042,E2 -5722.042} C_VEL
LIN {X 0,Y 502.775,Z 292.858,A -85,B 0,C 180,E1 -5725.032,E2 -5725.032} C_VEL
LIN {X 0,Y 502.748,Z 292.856,A -85,B 0,C 180,E1 -5727.912,E2 -5727.912} C_VEL
LIN {X 0,Y 502.749,Z 292.855,A -85,B 0,C 180,E1 -5730.707,E2 -5730.707} C_VEL
LIN {X 0,Y 502.761,Z 292.863,A -85,B 0,C 180,E1 -5733.46,E2 -5733.46} C_VEL
LIN {X 0,Y 502.748,Z 292.857,A -85,B 0,C 180,E1 -5736.084,E2 -5736.084} C_VEL
LIN {X 0,Y 502.767,Z 292.852,A -85,B 0,C 180,E1 -5738.688,E2 -5738.688} C_VEL
LIN {X 0,Y 502.792,Z 292.852,A -85,B 0,C 180,E1 -5741.246,E2 -5741.246} C_VEL
LIN {X 0,Y 502.782,Z 292.851,A -85,B 0,C 180,E1 -5744.682,E2 -5744.682} C_VEL
LIN {X 0,Y 502.86,Z 292.849,A -85,B 0,C 180,E1 -5748.043,E2 -5748.043} C_VEL
LIN {X 0,Y 502.826,Z 292.845,A -85,B 0,C 180,E1 -5751.156,E2 -5751.156} C_VEL
LIN {X 0,Y 502.857,Z 292.843,A -85,B 0,C 180,E1 -5753.58,E2 -5753.58} C_VEL
LIN {X 0,Y 502.851,Z 292.844,A -85,B 0,C 180,E1 -5756.795,E2 -5756.795} C_VEL
LIN {X 0,Y 502.887,Z 292.845,A -85,B 0,C 180,E1 -5758.398,E2 -5758.398} C_VEL
LIN {X 0,Y 502.979,Z 292.829,A -85,B 0,C 180,E1 -5760.8,E2 -5760.8} C_VEL
LIN {X 0,Y 503.001,Z 292.833,A -85,B 0,C 180,E1 -5762.402,E2 -5762.402} C_VEL
LIN {X 0,Y 502.909,Z 292.835,A -85,B 0,C 180,E1 -5765.614,E2 -5765.614} C_VEL
LIN {X 0,Y 502.861,Z 292.842,A -85,B 0,C 180,E1 -5768.034,E2 -5768.034} C_VEL
LIN {X 0,Y 502.863,Z 292.842,A -85,B 0,C 180,E1 -5771.283,E2 -5771.283} C_VEL
LIN {X 0,Y 502.819,Z 292.852,A -85,B 0,C 180,E1 -5774.572,E2 -5774.572} C_VEL
LIN {X 0,Y 502.802,Z 292.854,A -85,B 0,C 180,E1 -5777.069,E2 -5777.069} C_VEL
LIN {X 0,Y 502.809,Z 292.848,A -85,B 0,C 180,E1 -5779.6,E2 -5779.6} C_VEL
LIN {X 0,Y 502.793,Z 292.853,A -85,B 0,C 180,E1 -5782.702,E2 -5782.702} C_VEL
LIN {X 0,Y 502.777,Z 292.853,A -85,B 0,C 180,E1 -5785.679,E2 -5785.679} C_VEL
LIN {X 0,Y 502.828,Z 292.845,A -85,B 0,C 180,E1 -5788.373,E2 -5788.373} C_VEL
LIN {X 0,Y 502.784,Z 292.857,A -85,B 0,C 180,E1 -5791.499,E2 -5791.499} C_VEL
LIN {X 0,Y 502.796,Z 292.85,A -85,B 0,C 180,E1 -5793.995,E2 -5793.995} C_VEL
LIN {X 0,Y 502.757,Z 292.858,A -85,B 0,C 180,E1 -5797.176,E2 -5797.176} C_VEL
LIN {X 0,Y 502.781,Z 292.854,A -85,B 0,C 180,E1 -5800.016,E2 -5800.016} C_VEL
LIN {X 0,Y 502.797,Z 292.851,A -85,B 0,C 180,E1 -5802.2,E2 -5802.2} C_VEL
LIN {X 0,Y 502.78,Z 292.855,A -85,B 0,C 180,E1 -5805.471,E2 -5805.471} C_VEL
LIN {X 0,Y 502.79,Z 292.859,A -85,B 0,C 180,E1 -5807.861,E2 -5807.861} C_VEL
LIN {X 0,Y 502.796,Z 292.849,A -85,B 0,C 180,E1 -5811.025,E2 -5811.025} C_VEL
LIN {X 0,Y 502.767,Z 292.86,A -85,B 0,C 180,E1 -5814.171,E2 -5814.171} C_VEL
LIN {X 0,Y 502.83,Z 292.845,A -85,B 0,C 180,E1 -5816.994,E2 -5816.994} C_VEL
LIN {X 0,Y 502.812,Z 292.853,A -85,B 0,C 180,E1 -5820.066,E2 -5820.066} C_VEL
LIN {X 0,Y 502.822,Z 292.854,A -85,B 0,C 180,E1 -5822.534,E2 -5822.534} C_VEL
LIN {X 0,Y 502.812,Z 293.024,A -85,B 0,C 180,E1 -5825.396,E2 -5825.396} C_VEL
LIN {X 0,Y 504.494,Z 302.27,A -85,B 0,C 180,E1 -5827.043,E2 -5827.043} C_VEL
LIN {X 0,Y 503.996,Z 318.873,A -85,B 0,C 180,E1 -5829.811,E2 -5829.811} C_VEL
LIN {X 0,Y 503.475,Z 336.688,A -85,B 0,C 180,E1 -5832.746,E2 -5832.746} C_VEL
LIN {X 0,Y 503.254,Z 345.544,A -85,B 0,C 180,E1 -5834.194,E2 -5834.194} C_VEL
LIN {X 0,Y 505.376,Z 359.275,A -85,B 0,C 180,E1 -5834.461,E2 -5834.461} C_VEL
LIN {X 0,Y 504.876,Z 453.535,A -85,B 0,C 180,E1 -5835.824,E2 -5835.824} C_VEL
LIN {X 0,Y 504.603,Z 466.867,A -85,B 0,C 180,E1 -5836.176,E2 -5836.176} C_VEL
LIN {X 0,Y 504.238,Z 480.188,A -85,B 0,C 180,E1 -5836.705,E2 -5836.705} C_VEL
LIN {X 0,Y 503.911,Z 492.445,A -85,B 0,C 180,E1 -5837.381,E2 -5837.381} C_VEL
LIN {X 0,Y 503.545,Z 504.276,A -85,B 0,C 180,E1 -5838.223,E2 -5838.223} C_VEL
LIN {X 0,Y 503.177,Z 514.484,A -85,B 0,C 180,E1 -5839.132,E2 -5839.132} C_VEL
LIN {X 0,Y 502.851,Z 523.666,A -85,B 0,C 180,E1 -5840.143,E2 -5840.143} C_VEL
LIN {X 0,Y 502.575,Z 532.612,A -85,B 0,C 180,E1 -5841.355,E2 -5841.355} C_VEL
LIN {X 0,Y 502.347,Z 539.812,A -85,B 0,C 180,E1 -5842.565,E2 -5842.565} C_VEL
LIN {X 0,Y 502.234,Z 544.672,A -85,B 0,C 180,E1 -5843.573,E2 -5843.573} C_VEL
LIN {X 0,Y 502.174,Z 549.395,A -85,B 0,C 180,E1 -5844.781,E2 -5844.781} C_VEL
LIN {X 0,Y 502.138,Z 553.004,A -85,B 0,C 180,E1 -5845.988,E2 -5845.988} C_VEL
LIN {X 0,Y 502.12,Z 554.864,A -85,B 0,C 180,E1 -5846.791,E2 -5846.791} C_VEL
LIN {X 0,Y 502.091,Z 556.259,A -85,B 0,C 180,E1 -5847.594,E2 -5847.594} C_VEL
LIN {X 0,Y 501.99,Z 557.858,A -85,B 0,C 180,E1 -5849.198,E2 -5849.198} C_VEL
LIN {X 0,Y 501.981,Z 558.073,A -85,B 0,C 180,E1 -5850.001,E2 -5850.001} C_VEL
LIN {X 0,Y 502.036,Z 557.248,A -85,B 0,C 180,E1 -5851.605,E2 -5851.605} C_VEL
LIN {X 0,Y 502.091,Z 556.253,A -85,B 0,C 180,E1 -5852.407,E2 -5852.407} C_VEL
LIN {X 0,Y 502.12,Z 554.856,A -85,B 0,C 180,E1 -5853.21,E2 -5853.21} C_VEL
LIN {X 0,Y 502.102,Z 551.917,A -85,B 0,C 180,E1 -5854.416,E2 -5854.416} C_VEL
LIN {X 0,Y 502.21,Z 547.941,A -85,B 0,C 180,E1 -5855.622,E2 -5855.622} C_VEL
LIN {X 0,Y 502.33,Z 541.926,A -85,B 0,C 180,E1 -5857.012,E2 -5857.012} C_VEL
LIN {X 0,Y 502.477,Z 535.141,A -85,B 0,C 180,E1 -5858.243,E2 -5858.243} C_VEL
LIN {X 0,Y 502.746,Z 526.849,A -85,B 0,C 180,E1 -5859.454,E2 -5859.454} C_VEL
LIN {X 0,Y 502.99,Z 518.348,A -85,B 0,C 180,E1 -5860.466,E2 -5860.466} C_VEL
LIN {X 0,Y 503.412,Z 507.847,A -85,B 0,C 180,E1 -5861.475,E2 -5861.475} C_VEL
LIN {X 0,Y 503.709,Z 496.262,A -85,B 0,C 180,E1 -5862.371,E2 -5862.371} C_VEL
LIN {X 0,Y 504.132,Z 484.129,A -85,B 0,C 180,E1 -5863.094,E2 -5863.094} C_VEL
LIN {X 0,Y 504.512,Z 471.755,A -85,B 0,C 180,E1 -5863.648,E2 -5863.648} C_VEL
LIN {X 0,Y 504.746,Z 459.956,A -85,B 0,C 180,E1 -5864.026,E2 -5864.026} C_VEL
LIN {X 0,Y 504.922,Z 447.463,A -85,B 0,C 180,E1 -5864.278,E2 -5864.278} C_VEL
LIN {X 0,Y 505.296,Z 358.55,A -85,B 0,C 180,E1 -5865.551,E2 -5865.551} C_VEL
LIN {X 0,Y 503.231,Z 345.376,A -85,B 0,C 180,E1 -5865.822,E2 -5865.822} C_VEL
LIN {X 0,Y 503.734,Z 327.654,A -85,B 0,C 180,E1 -5868.717,E2 -5868.717} C_VEL
LIN {X 0,Y 504.27,Z 309.822,A -85,B 0,C 180,E1 -5871.675,E2 -5871.675} C_VEL
LIN {X 0,Y 504.374,Z 301.241,A -85,B 0,C 180,E1 -5873.125,E2 -5873.125} C_VEL
LIN {X 0,Y 502.785,Z 292.857,A -85,B 0,C 180,E1 -5874.642,E2 -5874.642} C_VEL
LIN {X 0,Y 502.827,Z 292.856,A -85,B 0,C 180,E1 -5877.468,E2 -5877.468} C_VEL
LIN {X 0,Y 502.81,Z 292.857,A -85,B 0,C 180,E1 -5880.211,E2 -5880.211} C_VEL
LIN {X 0,Y 502.834,Z 292.847,A -85,B 0,C 180,E1 -5883.031,E2 -5883.031} C_VEL
LIN {X 0,Y 502.77,Z 292.862,A -85,B 0,C 180,E1 -5885.952,E2 -5885.952} C_VEL
LIN {X 0,Y 502.798,Z 292.85,A -85,B 0,C 180,E1 -5888.977,E2 -5888.977} C_VEL
LIN {X 0,Y 502.805,Z 292.856,A -85,B 0,C 180,E1 -5892.199,E2 -5892.199} C_VEL
LIN {X 0,Y 502.787,Z 292.851,A -85,B 0,C 180,E1 -5895.47,E2 -5895.47} C_VEL
LIN {X 0,Y 502.796,Z 292.851,A -85,B 0,C 180,E1 -5897.861,E2 -5897.861} C_VEL
LIN {X 0,Y 502.802,Z 292.85,A -85,B 0,C 180,E1 -5901.024,E2 -5901.024} C_VEL
LIN {X 0,Y 502.772,Z 292.854,A -85,B 0,C 180,E1 -5904.17,E2 -5904.17} C_VEL
LIN {X 0,Y 502.834,Z 292.85,A -85,B 0,C 180,E1 -5906.993,E2 -5906.993} C_VEL
LIN {X 0,Y 502.815,Z 292.847,A -85,B 0,C 180,E1 -5910.065,E2 -5910.065} C_VEL
LIN {X 0,Y 502.844,Z 292.847,A -85,B 0,C 180,E1 -5913.444,E2 -5913.444} C_VEL
LIN {X 0,Y 502.787,Z 292.855,A -85,B 0,C 180,E1 -5916.959,E2 -5916.959} C_VEL
LIN {X 0,Y 502.837,Z 292.849,A -85,B 0,C 180,E1 -5919.548,E2 -5919.548} C_VEL
LIN {X 0,Y 502.823,Z 292.845,A -85,B 0,C 180,E1 -5922.092,E2 -5922.092} C_VEL
LIN {X 0,Y 502.843,Z 292.85,A -85,B 0,C 180,E1 -5925.429,E2 -5925.429} C_VEL
LIN {X 0,Y 502.877,Z 292.837,A -85,B 0,C 180,E1 -5928.717,E2 -5928.717} C_VEL
LIN {X 0,Y 502.88,Z 292.843,A -85,B 0,C 180,E1 -5931.966,E2 -5931.966} C_VEL
LIN {X 0,Y 502.929,Z 292.833,A -85,B 0,C 180,E1 -5934.387,E2 -5934.387} C_VEL
LIN {X 0,Y 503.019,Z 292.822,A -85,B 0,C 180,E1 -5937.598,E2 -5937.598} C_VEL
LIN {X 0,Y 503.028,Z 292.826,A -85,B 0,C 180,E1 -5940,E2 -5940} C_VEL
LIN {X 0,Y 503.019,Z 292.826,A -85,B 0,C 180,E1 -5942.402,E2 -5942.402} C_VEL
LIN {X 0,Y 502.926,Z 292.831,A -85,B 0,C 180,E1 -5945.614,E2 -5945.614} C_VEL
LIN {X 0,Y 502.869,Z 292.841,A -85,B 0,C 180,E1 -5948.844,E2 -5948.844} C_VEL
LIN {X 0,Y 502.847,Z 292.846,A -85,B 0,C 180,E1 -5952.102,E2 -5952.102} C_VEL
LIN {X 0,Y 502.85,Z 292.843,A -85,B 0,C 180,E1 -5955.4,E2 -5955.4} C_VEL
LIN {X 0,Y 502.827,Z 292.852,A -85,B 0,C 180,E1 -5958.752,E2 -5958.752} C_VEL
LIN {X 0,Y 502.785,Z 292.852,A -85,B 0,C 180,E1 -5961.311,E2 -5961.311} C_VEL
LIN {X 0,Y 502.775,Z 292.851,A -85,B 0,C 180,E1 -5963.915,E2 -5963.915} C_VEL
LIN {X 0,Y 502.837,Z 292.845,A -85,B 0,C 180,E1 -5966.568,E2 -5966.568} C_VEL
LIN {X 0,Y 502.816,Z 292.847,A -85,B 0,C 180,E1 -5969.935,E2 -5969.935} C_VEL
LIN {X 0,Y 502.832,Z 292.849,A -85,B 0,C 180,E1 -5973.032,E2 -5973.032} C_VEL
LIN {X 0,Y 502.77,Z 292.855,A -85,B 0,C 180,E1 -5975.952,E2 -5975.952} C_VEL
LIN {X 0,Y 502.804,Z 292.851,A -85,B 0,C 180,E1 -5978.976,E2 -5978.976} C_VEL
LIN {X 0,Y 502.807,Z 292.851,A -85,B 0,C 180,E1 -5982.199,E2 -5982.199} C_VEL
LIN {X 0,Y 502.789,Z 292.856,A -85,B 0,C 180,E1 -5985.47,E2 -5985.47} C_VEL
LIN {X 0,Y 502.799,Z 292.858,A -85,B 0,C 180,E1 -5987.861,E2 -5987.861} C_VEL
LIN {X 0,Y 502.796,Z 292.852,A -85,B 0,C 180,E1 -5991.023,E2 -5991.023} C_VEL
LIN {X 0,Y 502.772,Z 292.862,A -85,B 0,C 180,E1 -5994.17,E2 -5994.17} C_VEL
LIN {X 0,Y 502.796,Z 292.854,A -85,B 0,C 180,E1 -5997.213,E2 -5997.213} C_VEL
LIN {X 0,Y 502.501,Z 293.197,A -85,B 0,C 180,E1 -5997.656,E2 -5997.656} C_VEL
LIN {X 0,Y 501.303,Z 294.734,A -85,B 0,C 180,E1 -5998.292,E2 -5998.292} C_VEL
LIN {X 0,Y 499.666,Z 297.12,A -85,B 0,C 180,E1 -5998.889,E2 -5998.889} C_VEL
LIN {X 0,Y 497.527,Z 301.176,A -85,B 0,C 180,E1 -5999.667,E2 -5999.667} C_VEL
LIN {X 0,Y 496.61,Z 304.446,A -85,B 0,C 180,E1 -6000.252,E2 -6000.252} C_VEL
LIN {X 0,Y 496.534,Z 305.524,A -85,B 0,C 180,E1 -6000.45,E2 -6000.45} C_VEL
LIN {X 0,Y 496.292,Z 319.275,A -85,B 0,C 180,E1 -6003.007,E2 -6003.007} C_VEL
LIN {X 0,Y 498.674,Z 332.987,A -85,B 0,C 180,E1 -6003.298,E2 -6003.298} C_VEL
LIN {X 0,Y 498.001,Z 427.053,A -85,B 0,C 180,E1 -6004.684,E2 -6004.684} C_VEL
LIN {X 0,Y 497.771,Z 439.559,A -85,B 0,C 180,E1 -6005.023,E2 -6005.023} C_VEL
LIN {X 0,Y 497.49,Z 452.328,A -85,B 0,C 180,E1 -6005.537,E2 -6005.537} C_VEL
LIN {X 0,Y 497.11,Z 464.973,A -85,B 0,C 180,E1 -6006.238,E2 -6006.238} C_VEL
LIN {X 0,Y 496.74,Z 476.579,A -85,B 0,C 180,E1 -6007.077,E2 -6007.077} C_VEL
LIN {X 0,Y 496.283,Z 487.46,A -85,B 0,C 180,E1 -6008.068,E2 -6008.068} C_VEL
LIN {X 0,Y 495.995,Z 496.046,A -85,B 0,C 180,E1 -6009.036,E2 -6009.036} C_VEL
LIN {X 0,Y 495.617,Z 505.295,A -85,B 0,C 180,E1 -6010.319,E2 -6010.319} C_VEL
LIN {X 0,Y 495.387,Z 512.629,A -85,B 0,C 180,E1 -6011.599,E2 -6011.599} C_VEL
LIN {X 0,Y 495.202,Z 519.228,A -85,B 0,C 180,E1 -6013.085,E2 -6013.085} C_VEL
LIN {X 0,Y 495.112,Z 523.512,A -85,B 0,C 180,E1 -6014.353,E2 -6014.353} C_VEL
LIN {X 0,Y 495.057,Z 525.747,A -85,B 0,C 180,E1 -6015.194,E2 -6015.194} C_VEL
LIN {X 0,Y 494.961,Z 527.471,A -85,B 0,C 180,E1 -6016.031,E2 -6016.031} C_VEL
LIN {X 0,Y 494.937,Z 528.775,A -85,B 0,C 180,E1 -6016.867,E2 -6016.867} C_VEL
LIN {X 0,Y 495.011,Z 530.085,A -85,B 0,C 180,E1 -6018.42,E2 -6018.42} C_VEL
LIN {X 0,Y 494.951,Z 530.147,A -85,B 0,C 180,E1 -6019.362,E2 -6019.362} C_VEL
LIN {X 0,Y 494.93,Z 529.794,A -85,B 0,C 180,E1 -6020.188,E2 -6020.188} C_VEL
LIN {X 0,Y 494.949,Z 529.045,A -85,B 0,C 180,E1 -6021.013,E2 -6021.013} C_VEL
LIN {X 0,Y 494.996,Z 527.848,A -85,B 0,C 180,E1 -6021.837,E2 -6021.837} C_VEL
LIN {X 0,Y 495.047,Z 525.301,A -85,B 0,C 180,E1 -6023.069,E2 -6023.069} C_VEL
LIN {X 0,Y 495.175,Z 521.75,A -85,B 0,C 180,E1 -6024.298,E2 -6024.298} C_VEL
LIN {X 0,Y 495.256,Z 517.114,A -85,B 0,C 180,E1 -6025.523,E2 -6025.523} C_VEL
LIN {X 0,Y 495.402,Z 510.154,A -85,B 0,C 180,E1 -6026.95,E2 -6026.95} C_VEL
LIN {X 0,Y 495.686,Z 502.629,A -85,B 0,C 180,E1 -6028.171,E2 -6028.171} C_VEL
LIN {X 0,Y 496.041,Z 494.939,A -85,B 0,C 180,E1 -6029.188,E2 -6029.188} C_VEL
LIN {X 0,Y 496.264,Z 485.624,A -85,B 0,C 180,E1 -6030.202,E2 -6030.202} C_VEL
LIN {X 0,Y 496.692,Z 475.273,A -85,B 0,C 180,E1 -6031.114,E2 -6031.114} C_VEL
LIN {X 0,Y 497.15,Z 463.78,A -85,B 0,C 180,E1 -6031.923,E2 -6031.923} C_VEL
LIN {X 0,Y 497.483,Z 451.631,A -85,B 0,C 180,E1 -6032.58,E2 -6032.58} C_VEL
LIN {X 0,Y 497.763,Z 438.892,A -85,B 0,C 180,E1 -6033.085,E2 -6033.085} C_VEL
LIN {X 0,Y 497.947,Z 426.614,A -85,B 0,C 180,E1 -6033.413,E2 -6033.413} C_VEL
LIN {X 0,Y 498.611,Z 331.977,A -85,B 0,C 180,E1 -6034.8,E2 -6034.8} C_VEL
LIN {X 0,Y 496.226,Z 319.331,A -85,B 0,C 180,E1 -6035.078,E2 -6035.078} C_VEL
LIN {X 0,Y 496.691,Z 303.287,A -85,B 0,C 180,E1 -6038.134,E2 -6038.134} C_VEL
LIN {X 0,Y 496.547,Z 298.009,A -85,B 0,C 180,E1 -6039.161,E2 -6039.161} C_VEL
LIN {X 0,Y 495.813,Z 293.728,A -85,B 0,C 180,E1 -6040.05,E2 -6040.05} C_VEL
LIN {X 0,Y 495.79,Z 293.729,A -85,B 0,C 180,E1 -6042.276,E2 -6042.276} C_VEL
LIN {X 0,Y 495.806,Z 293.722,A -85,B 0,C 180,E1 -6045.442,E2 -6045.442} C_VEL
LIN {X 0,Y 495.769,Z 293.724,A -85,B 0,C 180,E1 -6049.028,E2 -6049.028} C_VEL
LIN {X 0,Y 495.741,Z 293.73,A -85,B 0,C 180,E1 -6051.628,E2 -6051.628} C_VEL
LIN {X 0,Y 495.713,Z 293.74,A -85,B 0,C 180,E1 -6054.276,E2 -6054.276} C_VEL
LIN {X 0,Y 495.728,Z 293.73,A -85,B 0,C 180,E1 -6056.978,E2 -6056.978} C_VEL
LIN {X 0,Y 495.743,Z 293.732,A -85,B 0,C 180,E1 -6060.142,E2 -6060.142} C_VEL
LIN {X 0,Y 495.749,Z 293.727,A -85,B 0,C 180,E1 -6063.236,E2 -6063.236} C_VEL
LIN {X 0,Y 495.701,Z 293.735,A -85,B 0,C 180,E1 -6066.085,E2 -6066.085} C_VEL
LIN {X 0,Y 495.736,Z 293.737,A -85,B 0,C 180,E1 -6068.764,E2 -6068.764} C_VEL
LIN {X 0,Y 495.719,Z 293.73,A -85,B 0,C 180,E1 -6071.784,E2 -6071.784} C_VEL
LIN {X 0,Y 495.726,Z 293.735,A -85,B 0,C 180,E1 -6075.141,E2 -6075.141} C_VEL
LIN {X 0,Y 495.718,Z 293.731,A -85,B 0,C 180,E1 -6078.214,E2 -6078.214} C_VEL
LIN {X 0,Y 495.733,Z 293.736,A -85,B 0,C 180,E1 -6081.235,E2 -6081.235} C_VEL
LIN {X 0,Y 495.722,Z 293.73,A -85,B 0,C 180,E1 -6084.46,E2 -6084.46} C_VEL
LIN {X 0,Y 495.717,Z 293.738,A -85,B 0,C 180,E1 -6087.401,E2 -6087.401} C_VEL
LIN {X 0,Y 495.691,Z 293.734,A -85,B 0,C 180,E1 -6090.248,E2 -6090.248} C_VEL
LIN {X 0,Y 495.712,Z 293.737,A -85,B 0,C 180,E1 -6093.274,E2 -6093.274} C_VEL
LIN {X 0,Y 495.696,Z 293.74,A -85,B 0,C 180,E1 -6095.722,E2 -6095.722} C_VEL
LIN {X 0,Y 495.729,Z 293.73,A -85,B 0,C 180,E1 -6098.37,E2 -6098.37} C_VEL
LIN {X 0,Y 495.752,Z 293.727,A -85,B 0,C 180,E1 -6100.97,E2 -6100.97} C_VEL
LIN {X 0,Y 495.751,Z 293.727,A -85,B 0,C 180,E1 -6104.575,E2 -6104.575} C_VEL
LIN {X 0,Y 495.812,Z 293.728,A -85,B 0,C 180,E1 -6107.969,E2 -6107.969} C_VEL
LIN {X 0,Y 495.783,Z 293.722,A -85,B 0,C 180,E1 -6111.029,E2 -6111.029} C_VEL
LIN {X 0,Y 495.808,Z 293.72,A -85,B 0,C 180,E1 -6113.489,E2 -6113.489} C_VEL
LIN {X 0,Y 495.709,Z 293.737,A -85,B 0,C 180,E1 -6115.935,E2 -6115.935} C_VEL
LIN {X 0,Y 495.97,Z 293.7,A -85,B 0,C 180,E1 -6117.563,E2 -6117.563} C_VEL
LIN {X 0,Y 495.931,Z 293.707,A -85,B 0,C 180,E1 -6120.812,E2 -6120.812} C_VEL
LIN {X 0,Y 495.969,Z 293.709,A -85,B 0,C 180,E1 -6122.436,E2 -6122.436} C_VEL
LIN {X 0,Y 495.865,Z 293.712,A -85,B 0,C 180,E1 -6125.694,E2 -6125.694} C_VEL
LIN {X 0,Y 495.818,Z 293.721,A -85,B 0,C 180,E1 -6128.149,E2 -6128.149} C_VEL
LIN {X 0,Y 495.839,Z 293.716,A -85,B 0,C 180,E1 -6131.445,E2 -6131.445} C_VEL
LIN {X 0,Y 495.769,Z 293.734,A -85,B 0,C 180,E1 -6134.783,E2 -6134.783} C_VEL
LIN {X 0,Y 495.748,Z 293.73,A -85,B 0,C 180,E1 -6137.32,E2 -6137.32} C_VEL
LIN {X 0,Y 495.757,Z 293.725,A -85,B 0,C 180,E1 -6139.891,E2 -6139.891} C_VEL
LIN {X 0,Y 495.749,Z 293.733,A -85,B 0,C 180,E1 -6142.86,E2 -6142.86} C_VEL
LIN {X 0,Y 495.744,Z 293.727,A -85,B 0,C 180,E1 -6146.07,E2 -6146.07} C_VEL
LIN {X 0,Y 495.76,Z 293.728,A -85,B 0,C 180,E1 -6148.816,E2 -6148.816} C_VEL
LIN {X 0,Y 495.747,Z 293.731,A -85,B 0,C 180,E1 -6151.726,E2 -6151.726} C_VEL
LIN {X 0,Y 495.76,Z 293.726,A -85,B 0,C 180,E1 -6154.694,E2 -6154.694} C_VEL
LIN {X 0,Y 495.715,Z 293.74,A -85,B 0,C 180,E1 -6157.563,E2 -6157.563} C_VEL
LIN {X 0,Y 495.752,Z 293.729,A -85,B 0,C 180,E1 -6160.048,E2 -6160.048} C_VEL
LIN {X 0,Y 495.711,Z 293.732,A -85,B 0,C 180,E1 -6162.885,E2 -6162.885} C_VEL
LIN {X 0,Y 495.719,Z 293.737,A -85,B 0,C 180,E1 -6165.999,E2 -6165.999} C_VEL
LIN {X 0,Y 495.734,Z 293.729,A -85,B 0,C 180,E1 -6168.71,E2 -6168.71} C_VEL
LIN {X 0,Y 495.745,Z 293.729,A -85,B 0,C 180,E1 -6171.409,E2 -6171.409} C_VEL
LIN {X 0,Y 495.741,Z 293.731,A -85,B 0,C 180,E1 -6174.463,E2 -6174.463} C_VEL
LIN {X 0,Y 495.765,Z 293.725,A -85,B 0,C 180,E1 -6177.407,E2 -6177.407} C_VEL
LIN {X 0,Y 495.763,Z 293.735,A -85,B 0,C 180,E1 -6180.254,E2 -6180.254} C_VEL
LIN {X 0,Y 495.804,Z 293.722,A -85,B 0,C 180,E1 -6183.256,E2 -6183.256} C_VEL
LIN {X 0,Y 495.756,Z 293.89,A -85,B 0,C 180,E1 -6185.227,E2 -6185.227} C_VEL
LIN {X 0,Y 497.488,Z 302.739,A -85,B 0,C 180,E1 -6186.829,E2 -6186.829} C_VEL
LIN {X 0,Y 497.088,Z 317.345,A -85,B 0,C 180,E1 -6189.302,E2 -6189.302} C_VEL
LIN {X 0,Y 496.57,Z 335.194,A -85,B 0,C 180,E1 -6192.285,E2 -6192.285} C_VEL
LIN {X 0,Y 496.244,Z 345.33,A -85,B 0,C 180,E1 -6193.965,E2 -6193.965} C_VEL
LIN {X 0,Y 498.533,Z 360.178,A -85,B 0,C 180,E1 -6194.261,E2 -6194.261} C_VEL
LIN {X 0,Y 498,Z 453.279,A -85,B 0,C 180,E1 -6195.624,E2 -6195.624} C_VEL
LIN {X 0,Y 497.683,Z 466.636,A -85,B 0,C 180,E1 -6195.98,E2 -6195.98} C_VEL
LIN {X 0,Y 497.335,Z 479.973,A -85,B 0,C 180,E1 -6196.517,E2 -6196.517} C_VEL
LIN {X 0,Y 497.02,Z 491.118,A -85,B 0,C 180,E1 -6197.13,E2 -6197.13} C_VEL
LIN {X 0,Y 496.574,Z 502.775,A -85,B 0,C 180,E1 -6197.951,E2 -6197.951} C_VEL
LIN {X 0,Y 496.23,Z 513.232,A -85,B 0,C 180,E1 -6198.875,E2 -6198.875} C_VEL
LIN {X 0,Y 495.862,Z 521.78,A -85,B 0,C 180,E1 -6199.796,E2 -6199.796} C_VEL
LIN {X 0,Y 495.617,Z 529.67,A -85,B 0,C 180,E1 -6200.821,E2 -6200.821} C_VEL
LIN {X 0,Y 495.342,Z 537.373,A -85,B 0,C 180,E1 -6202.049,E2 -6202.049} C_VEL
LIN {X 0,Y 495.163,Z 544.473,A -85,B 0,C 180,E1 -6203.481,E2 -6203.481} C_VEL
LIN {X 0,Y 495.106,Z 549.197,A -85,B 0,C 180,E1 -6204.707,E2 -6204.707} C_VEL
LIN {X 0,Y 495.031,Z 552.805,A -85,B 0,C 180,E1 -6205.93,E2 -6205.93} C_VEL
LIN {X 0,Y 495.041,Z 554.667,A -85,B 0,C 180,E1 -6206.745,E2 -6206.745} C_VEL
LIN {X 0,Y 494.997,Z 556.061,A -85,B 0,C 180,E1 -6207.559,E2 -6207.559} C_VEL
LIN {X 0,Y 494.962,Z 557.055,A -85,B 0,C 180,E1 -6208.373,E2 -6208.373} C_VEL
LIN {X 0,Y 494.899,Z 557.875,A -85,B 0,C 180,E1 -6210.001,E2 -6210.001} C_VEL
LIN {X 0,Y 494.962,Z 557.05,A -85,B 0,C 180,E1 -6211.628,E2 -6211.628} C_VEL
LIN {X 0,Y 494.997,Z 556.054,A -85,B 0,C 180,E1 -6212.442,E2 -6212.442} C_VEL
LIN {X 0,Y 495.042,Z 554.656,A -85,B 0,C 180,E1 -6213.256,E2 -6213.256} C_VEL
LIN {X 0,Y 495.008,Z 551.715,A -85,B 0,C 180,E1 -6214.479,E2 -6214.479} C_VEL
LIN {X 0,Y 495.126,Z 547.739,A -85,B 0,C 180,E1 -6215.703,E2 -6215.703} C_VEL
LIN {X 0,Y 495.256,Z 541.621,A -85,B 0,C 180,E1 -6217.133,E2 -6217.133} C_VEL
LIN {X 0,Y 495.425,Z 534.935,A -85,B 0,C 180,E1 -6218.361,E2 -6218.361} C_VEL
LIN {X 0,Y 495.716,Z 526.642,A -85,B 0,C 180,E1 -6219.59,E2 -6219.59} C_VEL
LIN {X 0,Y 495.983,Z 518.139,A -85,B 0,C 180,E1 -6220.615,E2 -6220.615} C_VEL
LIN {X 0,Y 496.429,Z 507.636,A -85,B 0,C 180,E1 -6221.639,E2 -6221.639} C_VEL
LIN {X 0,Y 496.76,Z 496.32,A -85,B 0,C 180,E1 -6222.527,E2 -6222.527} C_VEL
LIN {X 0,Y 497.203,Z 483.926,A -85,B 0,C 180,E1 -6223.28,E2 -6223.28} C_VEL
LIN {X 0,Y 497.614,Z 471.56,A -85,B 0,C 180,E1 -6223.841,E2 -6223.841} C_VEL
LIN {X 0,Y 497.911,Z 458.856,A -85,B 0,C 180,E1 -6224.249,E2 -6224.249} C_VEL
LIN {X 0,Y 498.058,Z 445.529,A -85,B 0,C 180,E1 -6224.506,E2 -6224.506} C_VEL
LIN {X 0,Y 498.41,Z 358.967,A -85,B 0,C 180,E1 -6225.765,E2 -6225.765} C_VEL
LIN {X 0,Y 496.249,Z 345.22,A -85,B 0,C 180,E1 -6226.046,E2 -6226.046} C_VEL
LIN {X 0,Y 496.737,Z 329.154,A -85,B 0,C 180,E1 -6228.713,E2 -6228.713} C_VEL
LIN {X 0,Y 497.333,Z 310.968,A -85,B 0,C 180,E1 -6231.775,E2 -6231.775} C_VEL
LIN {X 0,Y 497.491,Z 302.89,A -85,B 0,C 180,E1 -6233.159,E2 -6233.159} C_VEL
LIN {X 0,Y 495.736,Z 293.736,A -85,B 0,C 180,E1 -6234.862,E2 -6234.862} C_VEL
LIN {X 0,Y 495.786,Z 293.729,A -85,B 0,C 180,E1 -6236.976,E2 -6236.976} C_VEL
LIN {X 0,Y 495.768,Z 293.735,A -85,B 0,C 180,E1 -6239.747,E2 -6239.747} C_VEL
LIN {X 0,Y 495.77,Z 293.728,A -85,B 0,C 180,E1 -6242.594,E2 -6242.594} C_VEL
LIN {X 0,Y 495.747,Z 293.733,A -85,B 0,C 180,E1 -6245.538,E2 -6245.538} C_VEL
LIN {X 0,Y 495.762,Z 293.727,A -85,B 0,C 180,E1 -6248.768,E2 -6248.768} C_VEL
LIN {X 0,Y 495.752,Z 293.73,A -85,B 0,C 180,E1 -6251.782,E2 -6251.782} C_VEL
LIN {X 0,Y 495.739,Z 293.729,A -85,B 0,C 180,E1 -6255.141,E2 -6255.141} C_VEL
LIN {X 0,Y 495.752,Z 293.733,A -85,B 0,C 180,E1 -6258.218,E2 -6258.218} C_VEL
LIN {X 0,Y 495.75,Z 293.725,A -85,B 0,C 180,E1 -6261.408,E2 -6261.408} C_VEL
LIN {X 0,Y 495.746,Z 293.733,A -85,B 0,C 180,E1 -6264.462,E2 -6264.462} C_VEL
LIN {X 0,Y 495.768,Z 293.724,A -85,B 0,C 180,E1 -6267.406,E2 -6267.406} C_VEL
LIN {X 0,Y 495.763,Z 293.726,A -85,B 0,C 180,E1 -6270.253,E2 -6270.253} C_VEL
LIN {X 0,Y 495.775,Z 293.73,A -85,B 0,C 180,E1 -6273.262,E2 -6273.262} C_VEL
LIN {X 0,Y 495.74,Z 293.729,A -85,B 0,C 180,E1 -6276.612,E2 -6276.612} C_VEL
LIN {X 0,Y 495.78,Z 293.729,A -85,B 0,C 180,E1 -6279.324,E2 -6279.324} C_VEL
LIN {X 0,Y 495.782,Z 293.725,A -85,B 0,C 180,E1 -6281.829,E2 -6281.829} C_VEL
LIN {X 0,Y 495.825,Z 293.716,A -85,B 0,C 180,E1 -6284.549,E2 -6284.549} C_VEL
LIN {X 0,Y 495.829,Z 293.719,A -85,B 0,C 180,E1 -6287.965,E2 -6287.965} C_VEL
LIN {X 0,Y 495.833,Z 293.715,A -85,B 0,C 180,E1 -6291.03,E2 -6291.03} C_VEL
LIN {X 0,Y 495.858,Z 293.715,A -85,B 0,C 180,E1 -6293.49,E2 -6293.49} C_VEL
LIN {X 0,Y 495.719,Z 293.735,A -85,B 0,C 180,E1 -6295.935,E2 -6295.935} C_VEL
LIN {X 0,Y 495.986,Z 293.698,A -85,B 0,C 180,E1 -6297.564,E2 -6297.564} C_VEL
LIN {X 0,Y 495.942,Z 293.701,A -85,B 0,C 180,E1 -6300.812,E2 -6300.812} C_VEL
LIN {X 0,Y 495.986,Z 293.702,A -85,B 0,C 180,E1 -6302.437,E2 -6302.437} C_VEL
LIN {X 0,Y 495.881,Z 293.709,A -85,B 0,C 180,E1 -6305.694,E2 -6305.694} C_VEL
LIN {X 0,Y 495.838,Z 293.715,A -85,B 0,C 180,E1 -6308.97,E2 -6308.97} C_VEL
LIN {X 0,Y 495.83,Z 293.719,A -85,B 0,C 180,E1 -6312.035,E2 -6312.035} C_VEL
LIN {X 0,Y 495.825,Z 293.718,A -85,B 0,C 180,E1 -6315.452,E2 -6315.452} C_VEL
LIN {X 0,Y 495.78,Z 293.722,A -85,B 0,C 180,E1 -6318.237,E2 -6318.237} C_VEL
LIN {X 0,Y 495.776,Z 293.731,A -85,B 0,C 180,E1 -6320.757,E2 -6320.757} C_VEL
LIN {X 0,Y 495.743,Z 293.73,A -85,B 0,C 180,E1 -6323.388,E2 -6323.388} C_VEL
LIN {X 0,Y 495.777,Z 293.726,A -85,B 0,C 180,E1 -6326.738,E2 -6326.738} C_VEL
LIN {X 0,Y 495.765,Z 293.727,A -85,B 0,C 180,E1 -6329.747,E2 -6329.747} C_VEL
LIN {X 0,Y 495.768,Z 293.724,A -85,B 0,C 180,E1 -6332.595,E2 -6332.595} C_VEL
LIN {X 0,Y 495.747,Z 293.736,A -85,B 0,C 180,E1 -6335.538,E2 -6335.538} C_VEL
LIN {X 0,Y 495.766,Z 293.726,A -85,B 0,C 180,E1 -6338.768,E2 -6338.768} C_VEL
LIN {X 0,Y 495.753,Z 293.734,A -85,B 0,C 180,E1 -6341.782,E2 -6341.782} C_VEL
LIN {X 0,Y 495.741,Z 293.73,A -85,B 0,C 180,E1 -6345.141,E2 -6345.141} C_VEL
LIN {X 0,Y 495.747,Z 293.734,A -85,B 0,C 180,E1 -6348.218,E2 -6348.218} C_VEL
LIN {X 0,Y 495.748,Z 293.732,A -85,B 0,C 180,E1 -6351.408,E2 -6351.408} C_VEL
LIN {X 0,Y 495.746,Z 293.735,A -85,B 0,C 180,E1 -6354.462,E2 -6354.462} C_VEL
LIN {X 0,Y 495.765,Z 293.73,A -85,B 0,C 180,E1 -6357.405,E2 -6357.405} C_VEL
LIN {X 0,Y 495.774,Z 293.736,A -85,B 0,C 180,E1 -6358.195,E2 -6358.195} C_VEL
LIN {X 0,Y 496.606,Z 299.76,A -85,B 0,C 180,E1 -6359.371,E2 -6359.371} C_VEL
LIN {X 0,Y 496.534,Z 305.524,A -85,B 0,C 180,E1 -6360.45,E2 -6360.45} C_VEL
LIN {X 0,Y 495.85,Z 307.69,A -85,B 0,C 180,E1 -6360.827,E2 -6360.827} C_VEL
LIN {X 0,Y 492.98,Z 311.354,A -85,B 0,C 180,E1 -6361.391,E2 -6361.391} C_VEL
LIN {X 0,Y 490.071,Z 315.029,A -85,B 0,C 180,E1 -6361.961,E2 -6361.961} C_VEL
LIN {X 0,Y 489.347,Z 317.217,A -85,B 0,C 180,E1 -6362.343,E2 -6362.343} C_VEL
LIN {X 0,Y 489.342,Z 319.447,A -85,B 0,C 180,E1 -6362.763,E2 -6362.763} C_VEL
LIN {X 0,Y 491.796,Z 332.56,A -85,B 0,C 180,E1 -6363.053,E2 -6363.053} C_VEL
LIN {X 0,Y 491.168,Z 426.803,A -85,B 0,C 180,E1 -6364.462,E2 -6364.462} C_VEL
LIN {X 0,Y 490.905,Z 439.851,A -85,B 0,C 180,E1 -6364.819,E2 -6364.819} C_VEL
LIN {X 0,Y 490.6,Z 452.572,A -85,B 0,C 180,E1 -6365.34,E2 -6365.34} C_VEL
LIN {X 0,Y 490.235,Z 464.368,A -85,B 0,C 180,E1 -6365.997,E2 -6365.997} C_VEL
LIN {X 0,Y 489.836,Z 475.211,A -85,B 0,C 180,E1 -6366.773,E2 -6366.773} C_VEL
LIN {X 0,Y 489.385,Z 486.045,A -85,B 0,C 180,E1 -6367.742,E2 -6367.742} C_VEL
LIN {X 0,Y 489.044,Z 494.937,A -85,B 0,C 180,E1 -6368.723,E2 -6368.723} C_VEL
LIN {X 0,Y 488.752,Z 503.026,A -85,B 0,C 180,E1 -6369.811,E2 -6369.811} C_VEL
LIN {X 0,Y 488.401,Z 510.83,A -85,B 0,C 180,E1 -6371.108,E2 -6371.108} C_VEL
LIN {X 0,Y 488.208,Z 517.04,A -85,B 0,C 180,E1 -6372.403,E2 -6372.403} C_VEL
LIN {X 0,Y 488.05,Z 521.89,A -85,B 0,C 180,E1 -6373.691,E2 -6373.691} C_VEL
LIN {X 0,Y 487.996,Z 525.549,A -85,B 0,C 180,E1 -6374.975,E2 -6374.975} C_VEL
LIN {X 0,Y 487.897,Z 527.387,A -85,B 0,C 180,E1 -6375.825,E2 -6375.825} C_VEL
LIN {X 0,Y 487.859,Z 528.755,A -85,B 0,C 180,E1 -6376.673,E2 -6376.673} C_VEL
LIN {X 0,Y 487.853,Z 529.714,A -85,B 0,C 180,E1 -6377.52,E2 -6377.52} C_VEL
LIN {X 0,Y 487.932,Z 530.268,A -85,B 0,C 180,E1 -6378.366,E2 -6378.366} C_VEL
LIN {X 0,Y 487.865,Z 530.376,A -85,B 0,C 180,E1 -6379.206,E2 -6379.206} C_VEL
LIN {X 0,Y 487.843,Z 529.404,A -85,B 0,C 180,E1 -6380.881,E2 -6380.881} C_VEL
LIN {X 0,Y 487.913,Z 528.321,A -85,B 0,C 180,E1 -6381.718,E2 -6381.718} C_VEL
LIN {X 0,Y 487.929,Z 526.787,A -85,B 0,C 180,E1 -6382.551,E2 -6382.551} C_VEL
LIN {X 0,Y 488.015,Z 524.385,A -85,B 0,C 180,E1 -6383.561,E2 -6383.561} C_VEL
LIN {X 0,Y 488.079,Z 519.589,A -85,B 0,C 180,E1 -6385.043,E2 -6385.043} C_VEL
LIN {X 0,Y 488.303,Z 513.305,A -85,B 0,C 180,E1 -6386.493,E2 -6386.493} C_VEL
LIN {X 0,Y 488.477,Z 506.499,A -85,B 0,C 180,E1 -6387.732,E2 -6387.732} C_VEL
LIN {X 0,Y 488.923,Z 497.97,A -85,B 0,C 180,E1 -6388.97,E2 -6388.97} C_VEL
LIN {X 0,Y 489.171,Z 489.288,A -85,B 0,C 180,E1 -6389.999,E2 -6389.999} C_VEL
LIN {X 0,Y 489.573,Z 479.751,A -85,B 0,C 180,E1 -6390.925,E2 -6390.925} C_VEL
LIN {X 0,Y 490.028,Z 469.33,A -85,B 0,C 180,E1 -6391.746,E2 -6391.746} C_VEL
LIN {X 0,Y 490.411,Z 457.838,A -85,B 0,C 180,E1 -6392.463,E2 -6392.463} C_VEL
LIN {X 0,Y 490.697,Z 445.968,A -85,B 0,C 180,E1 -6393.027,E2 -6393.027} C_VEL
LIN {X 0,Y 490.974,Z 433.085,A -85,B 0,C 180,E1 -6393.461,E2 -6393.461} C_VEL
LIN {X 0,Y 491.184,Z 420.895,A -85,B 0,C 180,E1 -6393.717,E2 -6393.717} C_VEL
LIN {X 0,Y 491.646,Z 332.102,A -85,B 0,C 180,E1 -6395.022,E2 -6395.022} C_VEL
LIN {X 0,Y 489.299,Z 319.48,A -85,B 0,C 180,E1 -6395.305,E2 -6395.305} C_VEL
LIN {X 0,Y 489.794,Z 303.084,A -85,B 0,C 180,E1 -6398.457,E2 -6398.457} C_VEL
LIN {X 0,Y 489.359,Z 297.816,A -85,B 0,C 180,E1 -6399.506,E2 -6399.506} C_VEL
LIN {X 0,Y 488.747,Z 294.607,A -85,B 0,C 180,E1 -6400.197,E2 -6400.197} C_VEL
LIN {X 0,Y 488.741,Z 294.606,A -85,B 0,C 180,E1 -6402.456,E2 -6402.456} C_VEL
LIN {X 0,Y 488.765,Z 294.6,A -85,B 0,C 180,E1 -6405.548,E2 -6405.548} C_VEL
LIN {X 0,Y 488.746,Z 294.603,A -85,B 0,C 180,E1 -6408.442,E2 -6408.442} C_VEL
LIN {X 0,Y 488.708,Z 294.604,A -85,B 0,C 180,E1 -6411.07,E2 -6411.07} C_VEL
LIN {X 0,Y 488.67,Z 294.611,A -85,B 0,C 180,E1 -6413.746,E2 -6413.746} C_VEL
LIN {X 0,Y 488.695,Z 294.607,A -85,B 0,C 180,E1 -6416.92,E2 -6416.92} C_VEL
LIN {X 0,Y 488.704,Z 294.61,A -85,B 0,C 180,E1 -6420.22,E2 -6420.22} C_VEL
LIN {X 0,Y 488.708,Z 294.604,A -85,B 0,C 180,E1 -6423.479,E2 -6423.479} C_VEL
LIN {X 0,Y 488.662,Z 294.615,A -85,B 0,C 180,E1 -6426.351,E2 -6426.351} C_VEL
LIN {X 0,Y 488.683,Z 294.609,A -85,B 0,C 180,E1 -6429.255,E2 -6429.255} C_VEL
LIN {X 0,Y 488.663,Z 294.61,A -85,B 0,C 180,E1 -6431.593,E2 -6431.593} C_VEL
LIN {X 0,Y 488.691,Z 294.614,A -85,B 0,C 180,E1 -6434.802,E2 -6434.802} C_VEL
LIN {X 0,Y 488.643,Z 294.614,A -85,B 0,C 180,E1 -6437.469,E2 -6437.469} C_VEL
LIN {X 0,Y 488.698,Z 294.606,A -85,B 0,C 180,E1 -6439.673,E2 -6439.673} C_VEL
LIN {X 0,Y 488.644,Z 294.616,A -85,B 0,C 180,E1 -6442.838,E2 -6442.838} C_VEL
LIN {X 0,Y 488.702,Z 294.606,A -85,B 0,C 180,E1 -6445.884,E2 -6445.884} C_VEL
LIN {X 0,Y 488.65,Z 294.613,A -85,B 0,C 180,E1 -6448.817,E2 -6448.817} C_VEL
LIN {X 0,Y 488.677,Z 294.613,A -85,B 0,C 180,E1 -6451.667,E2 -6451.667} C_VEL
LIN {X 0,Y 488.683,Z 294.608,A -85,B 0,C 180,E1 -6454.96,E2 -6454.96} C_VEL
LIN {X 0,Y 488.686,Z 294.61,A -85,B 0,C 180,E1 -6458.042,E2 -6458.042} C_VEL
LIN {X 0,Y 488.716,Z 294.603,A -85,B 0,C 180,E1 -6460.685,E2 -6460.685} C_VEL
LIN {X 0,Y 488.673,Z 294.613,A -85,B 0,C 180,E1 -6464.142,E2 -6464.142} C_VEL
LIN {X 0,Y 488.693,Z 294.606,A -85,B 0,C 180,E1 -6466.697,E2 -6466.697} C_VEL
LIN {X 0,Y 488.774,Z 294.599,A -85,B 0,C 180,E1 -6468.387,E2 -6468.387} C_VEL
LIN {X 0,Y 488.746,Z 294.603,A -85,B 0,C 180,E1 -6471.732,E2 -6471.732} C_VEL
LIN {X 0,Y 488.8,Z 294.601,A -85,B 0,C 180,E1 -6474.223,E2 -6474.223} C_VEL
LIN {X 0,Y 488.938,Z 294.576,A -85,B 0,C 180,E1 -6477.528,E2 -6477.528} C_VEL
LIN {X 0,Y 488.883,Z 294.585,A -85,B 0,C 180,E1 -6480.824,E2 -6480.824} C_VEL
LIN {X 0,Y 488.936,Z 294.584,A -85,B 0,C 180,E1 -6482.471,E2 -6482.471} C_VEL
LIN {X 0,Y 488.824,Z 294.59,A -85,B 0,C 180,E1 -6485.776,E2 -6485.776} C_VEL
LIN {X 0,Y 488.764,Z 294.601,A -85,B 0,C 180,E1 -6488.267,E2 -6488.267} C_VEL
LIN {X 0,Y 488.794,Z 294.593,A -85,B 0,C 180,E1 -6491.613,E2 -6491.613} C_VEL
LIN {X 0,Y 488.745,Z 294.605,A -85,B 0,C 180,E1 -6495.001,E2 -6495.001} C_VEL
LIN {X 0,Y 488.736,Z 294.603,A -85,B 0,C 180,E1 -6498.443,E2 -6498.443} C_VEL
LIN {X 0,Y 488.697,Z 294.613,A -85,B 0,C 180,E1 -6501.071,E2 -6501.071} C_VEL
LIN {X 0,Y 488.66,Z 294.611,A -85,B 0,C 180,E1 -6503.747,E2 -6503.747} C_VEL
LIN {X 0,Y 488.738,Z 294.605,A -85,B 0,C 180,E1 -6506.934,E2 -6506.934} C_VEL
LIN {X 0,Y 488.713,Z 294.613,A -85,B 0,C 180,E1 -6509.271,E2 -6509.271} C_VEL
LIN {X 0,Y 488.695,Z 294.606,A -85,B 0,C 180,E1 -6512.148,E2 -6512.148} C_VEL
LIN {X 0,Y 488.708,Z 294.608,A -85,B 0,C 180,E1 -6515.116,E2 -6515.116} C_VEL
LIN {X 0,Y 488.67,Z 294.61,A -85,B 0,C 180,E1 -6518.201,E2 -6518.201} C_VEL
LIN {X 0,Y 488.712,Z 294.604,A -85,B 0,C 180,E1 -6520.345,E2 -6520.345} C_VEL
LIN {X 0,Y 488.672,Z 294.617,A -85,B 0,C 180,E1 -6523.656,E2 -6523.656} C_VEL
LIN {X 0,Y 488.672,Z 294.61,A -85,B 0,C 180,E1 -6526.345,E2 -6526.345} C_VEL
LIN {X 0,Y 488.698,Z 294.61,A -85,B 0,C 180,E1 -6529.674,E2 -6529.674} C_VEL
LIN {X 0,Y 488.666,Z 294.609,A -85,B 0,C 180,E1 -6532.841,E2 -6532.841} C_VEL
LIN {X 0,Y 488.727,Z 294.607,A -85,B 0,C 180,E1 -6535.888,E2 -6535.888} C_VEL
LIN {X 0,Y 488.688,Z 294.607,A -85,B 0,C 180,E1 -6538.821,E2 -6538.821} C_VEL
LIN {X 0,Y 488.739,Z 294.602,A -85,B 0,C 180,E1 -6541.672,E2 -6541.672} C_VEL
LIN {X 0,Y 488.707,Z 294.611,A -85,B 0,C 180,E1 -6544.443,E2 -6544.443} C_VEL
LIN {X 0,Y 488.713,Z 294.719,A -85,B 0,C 180,E1 -6545.05,E2 -6545.05} C_VEL
LIN {X 0,Y 490.572,Z 304.63,A -85,B 0,C 180,E1 -6546.865,E2 -6546.865} C_VEL
LIN {X 0,Y 490.035,Z 320.897,A -85,B 0,C 180,E1 -6549.649,E2 -6549.649} C_VEL
LIN {X 0,Y 489.483,Z 337.48,A -85,B 0,C 180,E1 -6552.452,E2 -6552.452} C_VEL
LIN {X 0,Y 489.282,Z 345.352,A -85,B 0,C 180,E1 -6553.747,E2 -6553.747} C_VEL
LIN {X 0,Y 491.667,Z 361.676,A -85,B 0,C 180,E1 -6554.066,E2 -6554.066} C_VEL
LIN {X 0,Y 491.106,Z 454.026,A -85,B 0,C 180,E1 -6555.445,E2 -6555.445} C_VEL
LIN {X 0,Y 490.782,Z 467.074,A -85,B 0,C 180,E1 -6555.805,E2 -6555.805} C_VEL
LIN {X 0,Y 490.418,Z 479.693,A -85,B 0,C 180,E1 -6556.323,E2 -6556.323} C_VEL
LIN {X 0,Y 490.055,Z 491.179,A -85,B 0,C 180,E1 -6556.964,E2 -6556.964} C_VEL
LIN {X 0,Y 489.602,Z 502.545,A -85,B 0,C 180,E1 -6557.777,E2 -6557.777} C_VEL
LIN {X 0,Y 489.224,Z 513.013,A -85,B 0,C 180,E1 -6558.713,E2 -6558.713} C_VEL
LIN {X 0,Y 488.84,Z 521.568,A -85,B 0,C 180,E1 -6559.648,E2 -6559.648} C_VEL
LIN {X 0,Y 488.557,Z 529.462,A -85,B 0,C 180,E1 -6560.687,E2 -6560.687} C_VEL
LIN {X 0,Y 488.276,Z 537.171,A -85,B 0,C 180,E1 -6561.933,E2 -6561.933} C_VEL
LIN {X 0,Y 488.1,Z 544.274,A -85,B 0,C 180,E1 -6563.386,E2 -6563.386} C_VEL
LIN {X 0,Y 488.018,Z 548.998,A -85,B 0,C 180,E1 -6564.629,E2 -6564.629} C_VEL
LIN {X 0,Y 487.927,Z 552.606,A -85,B 0,C 180,E1 -6565.871,E2 -6565.871} C_VEL
LIN {X 0,Y 487.964,Z 554.469,A -85,B 0,C 180,E1 -6566.698,E2 -6566.698} C_VEL
LIN {X 0,Y 487.89,Z 556.858,A -85,B 0,C 180,E1 -6568.35,E2 -6568.35} C_VEL
LIN {X 0,Y 487.82,Z 557.677,A -85,B 0,C 180,E1 -6570.001,E2 -6570.001} C_VEL
LIN {X 0,Y 487.89,Z 556.851,A -85,B 0,C 180,E1 -6571.651,E2 -6571.651} C_VEL
LIN {X 0,Y 487.964,Z 554.457,A -85,B 0,C 180,E1 -6573.303,E2 -6573.303} C_VEL
LIN {X 0,Y 487.92,Z 551.514,A -85,B 0,C 180,E1 -6574.544,E2 -6574.544} C_VEL
LIN {X 0,Y 488.024,Z 547.536,A -85,B 0,C 180,E1 -6575.786,E2 -6575.786} C_VEL
LIN {X 0,Y 488.181,Z 541.418,A -85,B 0,C 180,E1 -6577.237,E2 -6577.237} C_VEL
LIN {X 0,Y 488.36,Z 534.734,A -85,B 0,C 180,E1 -6578.483,E2 -6578.483} C_VEL
LIN {X 0,Y 488.684,Z 526.445,A -85,B 0,C 180,E1 -6579.729,E2 -6579.729} C_VEL
LIN {X 0,Y 488.993,Z 517.947,A -85,B 0,C 180,E1 -6580.769,E2 -6580.769} C_VEL
LIN {X 0,Y 489.45,Z 507.456,A -85,B 0,C 180,E1 -6581.807,E2 -6581.807} C_VEL
LIN {X 0,Y 489.828,Z 495.748,A -85,B 0,C 180,E1 -6582.738,E2 -6582.738} C_VEL
LIN {X 0,Y 490.279,Z 483.797,A -85,B 0,C 180,E1 -6583.471,E2 -6583.471} C_VEL
LIN {X 0,Y 490.733,Z 471.467,A -85,B 0,C 180,E1 -6584.039,E2 -6584.039} C_VEL
LIN {X 0,Y 491.018,Z 459.741,A -85,B 0,C 180,E1 -6584.427,E2 -6584.427} C_VEL
LIN {X 0,Y 491.182,Z 447.446,A -85,B 0,C 180,E1 -6584.687,E2 -6584.687} C_VEL
LIN {X 0,Y 491.621,Z 359.938,A -85,B 0,C 180,E1 -6585.979,E2 -6585.979} C_VEL
LIN {X 0,Y 489.277,Z 344.903,A -85,B 0,C 180,E1 -6586.309,E2 -6586.309} C_VEL
LIN {X 0,Y 489.78,Z 328.386,A -85,B 0,C 180,E1 -6589.098,E2 -6589.098} C_VEL
LIN {X 0,Y 490.415,Z 310.865,A -85,B 0,C 180,E1 -6592.098,E2 -6592.098} C_VEL
LIN {X 0,Y 490.488,Z 303.798,A -85,B 0,C 180,E1 -6593.333,E2 -6593.333} C_VEL
LIN {X 0,Y 488.7,Z 294.613,A -85,B 0,C 180,E1 -6595.103,E2 -6595.103} C_VEL
LIN {X 0,Y 488.733,Z 294.611,A -85,B 0,C 180,E1 -6597.398,E2 -6597.398} C_VEL
LIN {X 0,Y 488.711,Z 294.612,A -85,B 0,C 180,E1 -6600.363,E2 -6600.363} C_VEL
LIN {X 0,Y 488.737,Z 294.607,A -85,B 0,C 180,E1 -6603.484,E2 -6603.484} C_VEL
LIN {X 0,Y 488.675,Z 294.615,A -85,B 0,C 180,E1 -6606.353,E2 -6606.353} C_VEL
LIN {X 0,Y 488.699,Z 294.606,A -85,B 0,C 180,E1 -6609.255,E2 -6609.255} C_VEL
LIN {X 0,Y 488.699,Z 294.607,A -85,B 0,C 180,E1 -6611.599,E2 -6611.599} C_VEL
LIN {X 0,Y 488.703,Z 294.609,A -85,B 0,C 180,E1 -6614.803,E2 -6614.803} C_VEL
LIN {X 0,Y 488.69,Z 294.607,A -85,B 0,C 180,E1 -6617.474,E2 -6617.474} C_VEL
LIN {X 0,Y 488.702,Z 294.61,A -85,B 0,C 180,E1 -6620.746,E2 -6620.746} C_VEL
LIN {X 0,Y 488.67,Z 294.609,A -85,B 0,C 180,E1 -6623.867,E2 -6623.867} C_VEL
LIN {X 0,Y 488.739,Z 294.607,A -85,B 0,C 180,E1 -6626.877,E2 -6626.877} C_VEL
LIN {X 0,Y 488.724,Z 294.603,A -85,B 0,C 180,E1 -6629.781,E2 -6629.781} C_VEL
LIN {X 0,Y 488.726,Z 294.611,A -85,B 0,C 180,E1 -6633.072,E2 -6633.072} C_VEL
LIN {X 0,Y 488.67,Z 294.608,A -85,B 0,C 180,E1 -6636.253,E2 -6636.253} C_VEL
LIN {X 0,Y 488.747,Z 294.605,A -85,B 0,C 180,E1 -6639.176,E2 -6639.176} C_VEL
LIN {X 0,Y 488.75,Z 294.603,A -85,B 0,C 180,E1 -6641.632,E2 -6641.632} C_VEL
LIN {X 0,Y 488.762,Z 294.598,A -85,B 0,C 180,E1 -6645,E2 -6645} C_VEL
LIN {X 0,Y 488.806,Z 294.591,A -85,B 0,C 180,E1 -6648.388,E2 -6648.388} C_VEL
LIN {X 0,Y 488.785,Z 294.598,A -85,B 0,C 180,E1 -6651.733,E2 -6651.733} C_VEL
LIN {X 0,Y 488.844,Z 294.589,A -85,B 0,C 180,E1 -6654.224,E2 -6654.224} C_VEL
LIN {X 0,Y 488.953,Z 294.573,A -85,B 0,C 180,E1 -6657.529,E2 -6657.529} C_VEL
LIN {X 0,Y 488.97,Z 294.576,A -85,B 0,C 180,E1 -6660,E2 -6660} C_VEL
LIN {X 0,Y 488.953,Z 294.577,A -85,B 0,C 180,E1 -6662.472,E2 -6662.472} C_VEL
LIN {X 0,Y 488.839,Z 294.587,A -85,B 0,C 180,E1 -6665.776,E2 -6665.776} C_VEL
LIN {X 0,Y 488.787,Z 294.601,A -85,B 0,C 180,E1 -6668.267,E2 -6668.267} C_VEL
LIN {X 0,Y 488.806,Z 294.592,A -85,B 0,C 180,E1 -6671.613,E2 -6671.613} C_VEL
LIN {X 0,Y 488.763,Z 294.602,A -85,B 0,C 180,E1 -6675.001,E2 -6675.001} C_VEL
LIN {X 0,Y 488.748,Z 294.6,A -85,B 0,C 180,E1 -6678.443,E2 -6678.443} C_VEL
LIN {X 0,Y 488.709,Z 294.608,A -85,B 0,C 180,E1 -6681.071,E2 -6681.071} C_VEL
LIN {X 0,Y 488.676,Z 294.608,A -85,B 0,C 180,E1 -6683.747,E2 -6683.747} C_VEL
LIN {X 0,Y 488.719,Z 294.603,A -85,B 0,C 180,E1 -6686.474,E2 -6686.474} C_VEL
LIN {X 0,Y 488.712,Z 294.61,A -85,B 0,C 180,E1 -6689.271,E2 -6689.271} C_VEL
LIN {X 0,Y 488.704,Z 294.604,A -85,B 0,C 180,E1 -6692.147,E2 -6692.147} C_VEL
LIN {X 0,Y 488.716,Z 294.607,A -85,B 0,C 180,E1 -6695.116,E2 -6695.116} C_VEL
LIN {X 0,Y 488.68,Z 294.61,A -85,B 0,C 180,E1 -6698.2,E2 -6698.2} C_VEL
LIN {X 0,Y 488.722,Z 294.604,A -85,B 0,C 180,E1 -6700.345,E2 -6700.345} C_VEL
LIN {X 0,Y 488.681,Z 294.616,A -85,B 0,C 180,E1 -6703.656,E2 -6703.656} C_VEL
LIN {X 0,Y 488.678,Z 294.612,A -85,B 0,C 180,E1 -6706.344,E2 -6706.344} C_VEL
LIN {X 0,Y 488.707,Z 294.61,A -85,B 0,C 180,E1 -6709.674,E2 -6709.674} C_VEL
LIN {X 0,Y 488.67,Z 294.613,A -85,B 0,C 180,E1 -6712.84,E2 -6712.84} C_VEL
LIN {X 0,Y 488.722,Z 294.609,A -85,B 0,C 180,E1 -6715.886,E2 -6715.886} C_VEL
LIN {X 0,Y 488.755,Z 294.703,A -85,B 0,C 180,E1 -6718.037,E2 -6718.037} C_VEL
LIN {X 0,Y 489.654,Z 300.672,A -85,B 0,C 180,E1 -6719.222,E2 -6719.222} C_VEL
LIN {X 0,Y 489.408,Z 315.093,A -85,B 0,C 180,E1 -6721.946,E2 -6721.946} C_VEL
LIN {X 0,Y 489.347,Z 317.217,A -85,B 0,C 180,E1 -6722.343,E2 -6722.343} C_VEL
LIN {X 0,Y 488.834,Z 319.125,A -85,B 0,C 180,E1 -6722.56,E2 -6722.56} C_VEL
LIN {X 0,Y 487.324,Z 322.337,A -85,B 0,C 180,E1 -6722.703,E2 -6722.703} C_VEL
LIN {X 0,Y 484.319,Z 328.839,A -85,B 0,C 180,E1 -6722.724,E2 -6722.724} C_VEL
LIN {X 0,Y 483.554,Z 332.998,A -85,B 0,C 180,E1 -6722.752,E2 -6722.752} C_VEL
LIN {X 0,Y 484.039,Z 339.464,A -85,B 0,C 180,E1 -6722.867,E2 -6722.867} C_VEL
LIN {X 0,Y 484.91,Z 345.944,A -85,B 0,C 180,E1 -6723.006,E2 -6723.006} C_VEL
LIN {X 0,Y 484.961,Z 348.13,A -85,B 0,C 180,E1 -6723.042,E2 -6723.042} C_VEL
LIN {X 0,Y 484.34,Z 427.275,A -85,B 0,C 180,E1 -6724.246,E2 -6724.246} C_VEL
LIN {X 0,Y 484.072,Z 439.483,A -85,B 0,C 180,E1 -6724.583,E2 -6724.583} C_VEL
LIN {X 0,Y 483.752,Z 451.742,A -85,B 0,C 180,E1 -6725.082,E2 -6725.082} C_VEL
LIN {X 0,Y 483.383,Z 463.826,A -85,B 0,C 180,E1 -6725.749,E2 -6725.749} C_VEL
LIN {X 0,Y 482.923,Z 475.241,A -85,B 0,C 180,E1 -6726.571,E2 -6726.571} C_VEL
LIN {X 0,Y 482.476,Z 485.741,A -85,B 0,C 180,E1 -6727.519,E2 -6727.519} C_VEL
LIN {X 0,Y 482.04,Z 495.616,A -85,B 0,C 180,E1 -6728.623,E2 -6728.623} C_VEL
LIN {X 0,Y 481.711,Z 503.597,A -85,B 0,C 180,E1 -6729.726,E2 -6729.726} C_VEL
LIN {X 0,Y 481.36,Z 511.33,A -85,B 0,C 180,E1 -6731.043,E2 -6731.043} C_VEL
LIN {X 0,Y 481.157,Z 516.544,A -85,B 0,C 180,E1 -6732.137,E2 -6732.137} C_VEL
LIN {X 0,Y 481.012,Z 521.543,A -85,B 0,C 180,E1 -6733.446,E2 -6733.446} C_VEL
LIN {X 0,Y 480.918,Z 525.34,A -85,B 0,C 180,E1 -6734.749,E2 -6734.749} C_VEL
LIN {X 0,Y 480.847,Z 527.28,A -85,B 0,C 180,E1 -6735.613,E2 -6735.613} C_VEL
LIN {X 0,Y 480.766,Z 528.74,A -85,B 0,C 180,E1 -6736.473,E2 -6736.473} C_VEL
LIN {X 0,Y 480.771,Z 529.76,A -85,B 0,C 180,E1 -6737.333,E2 -6737.333} C_VEL
LIN {X 0,Y 480.844,Z 530.449,A -85,B 0,C 180,E1 -6738.316,E2 -6738.316} C_VEL
LIN {X 0,Y 480.742,Z 530.375,A -85,B 0,C 180,E1 -6739.896,E2 -6739.896} C_VEL
LIN {X 0,Y 480.809,Z 528.741,A -85,B 0,C 180,E1 -6741.594,E2 -6741.594} C_VEL
LIN {X 0,Y 480.84,Z 527.319,A -85,B 0,C 180,E1 -6742.441,E2 -6742.441} C_VEL
LIN {X 0,Y 480.925,Z 524.693,A -85,B 0,C 180,E1 -6743.579,E2 -6743.579} C_VEL
LIN {X 0,Y 480.997,Z 520.377,A -85,B 0,C 180,E1 -6744.97,E2 -6744.97} C_VEL
LIN {X 0,Y 481.236,Z 515.24,A -85,B 0,C 180,E1 -6746.231,E2 -6746.231} C_VEL
LIN {X 0,Y 481.366,Z 508.816,A -85,B 0,C 180,E1 -6747.489,E2 -6747.489} C_VEL
LIN {X 0,Y 481.802,Z 500.81,A -85,B 0,C 180,E1 -6748.746,E2 -6748.746} C_VEL
LIN {X 0,Y 482.075,Z 492.689,A -85,B 0,C 180,E1 -6749.791,E2 -6749.791} C_VEL
LIN {X 0,Y 482.504,Z 482.778,A -85,B 0,C 180,E1 -6750.834,E2 -6750.834} C_VEL
LIN {X 0,Y 482.925,Z 472.979,A -85,B 0,C 180,E1 -6751.667,E2 -6751.667} C_VEL
LIN {X 0,Y 483.409,Z 460.618,A -85,B 0,C 180,E1 -6752.499,E2 -6752.499} C_VEL
LIN {X 0,Y 483.751,Z 448.512,A -85,B 0,C 180,E1 -6753.122,E2 -6753.122} C_VEL
LIN {X 0,Y 484.044,Z 435.745,A -85,B 0,C 180,E1 -6753.589,E2 -6753.589} C_VEL
LIN {X 0,Y 484.265,Z 422.213,A -85,B 0,C 180,E1 -6753.9,E2 -6753.9} C_VEL
LIN {X 0,Y 484.859,Z 333.415,A -85,B 0,C 180,E1 -6755.223,E2 -6755.223} C_VEL
LIN {X 0,Y 482.298,Z 319.608,A -85,B 0,C 180,E1 -6755.539,E2 -6755.539} C_VEL
LIN {X 0,Y 482.837,Z 303.951,A -85,B 0,C 180,E1 -6758.58,E2 -6758.58} C_VEL
LIN {X 0,Y 482.301,Z 298.667,A -85,B 0,C 180,E1 -6759.646,E2 -6759.646} C_VEL
LIN {X 0,Y 481.721,Z 295.481,A -85,B 0,C 180,E1 -6760.348,E2 -6760.348} C_VEL
LIN {X 0,Y 481.685,Z 295.484,A -85,B 0,C 180,E1 -6762.641,E2 -6762.641} C_VEL
LIN {X 0,Y 481.716,Z 295.479,A -85,B 0,C 180,E1 -6765.653,E2 -6765.653} C_VEL
LIN {X 0,Y 481.706,Z 295.477,A -85,B 0,C 180,E1 -6768.721,E2 -6768.721} C_VEL
LIN {X 0,Y 481.646,Z 295.484,A -85,B 0,C 180,E1 -6771.394,E2 -6771.394} C_VEL
LIN {X 0,Y 481.648,Z 295.491,A -85,B 0,C 180,E1 -6774.114,E2 -6774.114} C_VEL
LIN {X 0,Y 481.65,Z 295.483,A -85,B 0,C 180,E1 -6777.115,E2 -6777.115} C_VEL
LIN {X 0,Y 481.654,Z 295.483,A -85,B 0,C 180,E1 -6779.742,E2 -6779.742} C_VEL
LIN {X 0,Y 481.65,Z 295.49,A -85,B 0,C 180,E1 -6782.675,E2 -6782.675} C_VEL
LIN {X 0,Y 481.623,Z 295.486,A -85,B 0,C 180,E1 -6785.709,E2 -6785.709} C_VEL
LIN {X 0,Y 481.652,Z 295.49,A -85,B 0,C 180,E1 -6788.86,E2 -6788.86} C_VEL
LIN {X 0,Y 481.616,Z 295.487,A -85,B 0,C 180,E1 -6791.907,E2 -6791.907} C_VEL
LIN {X 0,Y 481.645,Z 295.487,A -85,B 0,C 180,E1 -6794.458,E2 -6794.458} C_VEL
LIN {X 0,Y 481.607,Z 295.496,A -85,B 0,C 180,E1 -6796.855,E2 -6796.855} C_VEL
LIN {X 0,Y 481.65,Z 295.483,A -85,B 0,C 180,E1 -6800.056,E2 -6800.056} C_VEL
LIN {X 0,Y 481.602,Z 295.495,A -85,B 0,C 180,E1 -6803.378,E2 -6803.378} C_VEL
LIN {X 0,Y 481.664,Z 295.481,A -85,B 0,C 180,E1 -6806.326,E2 -6806.326} C_VEL
LIN {X 0,Y 481.603,Z 295.497,A -85,B 0,C 180,E1 -6809.425,E2 -6809.425} C_VEL
LIN {X 0,Y 481.634,Z 295.486,A -85,B 0,C 180,E1 -6812.164,E2 -6812.164} C_VEL
LIN {X 0,Y 481.657,Z 295.484,A -85,B 0,C 180,E1 -6814.966,E2 -6814.966} C_VEL
LIN {X 0,Y 481.638,Z 295.492,A -85,B 0,C 180,E1 -6817.704,E2 -6817.704} C_VEL
LIN {X 0,Y 481.683,Z 295.48,A -85,B 0,C 180,E1 -6820.392,E2 -6820.392} C_VEL
LIN {X 0,Y 481.601,Z 295.49,A -85,B 0,C 180,E1 -6823.03,E2 -6823.03} C_VEL
LIN {X 0,Y 481.638,Z 295.49,A -85,B 0,C 180,E1 -6825.637,E2 -6825.637} C_VEL
LIN {X 0,Y 481.725,Z 295.479,A -85,B 0,C 180,E1 -6828.214,E2 -6828.214} C_VEL
LIN {X 0,Y 481.705,Z 295.479,A -85,B 0,C 180,E1 -6831.61,E2 -6831.61} C_VEL
LIN {X 0,Y 481.762,Z 295.479,A -85,B 0,C 180,E1 -6834.139,E2 -6834.139} C_VEL
LIN {X 0,Y 481.904,Z 295.452,A -85,B 0,C 180,E1 -6837.492,E2 -6837.492} C_VEL
LIN {X 0,Y 481.836,Z 295.462,A -85,B 0,C 180,E1 -6840.836,E2 -6840.836} C_VEL
LIN {X 0,Y 481.902,Z 295.459,A -85,B 0,C 180,E1 -6842.507,E2 -6842.507} C_VEL
LIN {X 0,Y 481.785,Z 295.467,A -85,B 0,C 180,E1 -6845.861,E2 -6845.861} C_VEL
LIN {X 0,Y 481.719,Z 295.48,A -85,B 0,C 180,E1 -6848.389,E2 -6848.389} C_VEL
LIN {X 0,Y 481.74,Z 295.472,A -85,B 0,C 180,E1 -6851.785,E2 -6851.785} C_VEL
LIN {X 0,Y 481.729,Z 295.476,A -85,B 0,C 180,E1 -6855.225,E2 -6855.225} C_VEL
LIN {X 0,Y 481.698,Z 295.483,A -85,B 0,C 180,E1 -6858.722,E2 -6858.722} C_VEL
LIN {X 0,Y 481.636,Z 295.488,A -85,B 0,C 180,E1 -6861.395,E2 -6861.395} C_VEL
LIN {X 0,Y 481.639,Z 295.484,A -85,B 0,C 180,E1 -6864.115,E2 -6864.115} C_VEL
LIN {X 0,Y 481.706,Z 295.484,A -85,B 0,C 180,E1 -6867.132,E2 -6867.132} C_VEL
LIN {X 0,Y 481.669,Z 295.483,A -85,B 0,C 180,E1 -6869.742,E2 -6869.742} C_VEL
LIN {X 0,Y 481.664,Z 295.482,A -85,B 0,C 180,E1 -6872.675,E2 -6872.675} C_VEL
LIN {X 0,Y 481.625,Z 295.492,A -85,B 0,C 180,E1 -6875.711,E2 -6875.711} C_VEL
LIN {X 0,Y 481.663,Z 295.482,A -85,B 0,C 180,E1 -6878.86,E2 -6878.86} C_VEL
LIN {X 0,Y 481.641,Z 295.49,A -85,B 0,C 180,E1 -6881.913,E2 -6881.913} C_VEL
LIN {X 0,Y 481.648,Z 295.484,A -85,B 0,C 180,E1 -6884.459,E2 -6884.459} C_VEL
LIN {X 0,Y 481.638,Z 295.494,A -85,B 0,C 180,E1 -6887.84,E2 -6887.84} C_VEL
LIN {X 0,Y 481.655,Z 295.483,A -85,B 0,C 180,E1 -6890.655,E2 -6890.655} C_VEL
LIN {X 0,Y 481.618,Z 295.488,A -85,B 0,C 180,E1 -6893.378,E2 -6893.378} C_VEL
LIN {X 0,Y 481.707,Z 295.482,A -85,B 0,C 180,E1 -6896.331,E2 -6896.331} C_VEL
LIN {X 0,Y 481.647,Z 295.484,A -85,B 0,C 180,E1 -6899.419,E2 -6899.419} C_VEL
LIN {X 0,Y 481.689,Z 295.486,A -85,B 0,C 180,E1 -6902.168,E2 -6902.168} C_VEL
LIN {X 0,Y 481.672,Z 295.529,A -85,B 0,C 180,E1 -6904.866,E2 -6904.866} C_VEL
LIN {X 0,Y 483.627,Z 306.496,A -85,B 0,C 180,E1 -6906.9,E2 -6906.9} C_VEL
LIN {X 0,Y 482.952,Z 324.436,A -85,B 0,C 180,E1 -6910.004,E2 -6910.004} C_VEL
LIN {X 0,Y 482.362,Z 341.02,A -85,B 0,C 180,E1 -6912.841,E2 -6912.841} C_VEL
LIN {X 0,Y 482.261,Z 345.07,A -85,B 0,C 180,E1 -6913.515,E2 -6913.515} C_VEL
LIN {X 0,Y 484.831,Z 362.771,A -85,B 0,C 180,E1 -6913.865,E2 -6913.865} C_VEL
LIN {X 0,Y 484.238,Z 453.425,A -85,B 0,C 180,E1 -6915.234,E2 -6915.234} C_VEL
LIN {X 0,Y 483.88,Z 466.613,A -85,B 0,C 180,E1 -6915.599,E2 -6915.599} C_VEL
LIN {X 0,Y 483.521,Z 479.312,A -85,B 0,C 180,E1 -6916.124,E2 -6916.124} C_VEL
LIN {X 0,Y 483.139,Z 490.597,A -85,B 0,C 180,E1 -6916.756,E2 -6916.756} C_VEL
LIN {X 0,Y 482.629,Z 502.258,A -85,B 0,C 180,E1 -6917.598,E2 -6917.598} C_VEL
LIN {X 0,Y 482.193,Z 512.748,A -85,B 0,C 180,E1 -6918.546,E2 -6918.546} C_VEL
LIN {X 0,Y 481.818,Z 521.322,A -85,B 0,C 180,E1 -6919.495,E2 -6919.495} C_VEL
LIN {X 0,Y 481.503,Z 529.23,A -85,B 0,C 180,E1 -6920.55,E2 -6920.55} C_VEL
LIN {X 0,Y 481.226,Z 536.952,A -85,B 0,C 180,E1 -6921.814,E2 -6921.814} C_VEL
LIN {X 0,Y 481.019,Z 544.063,A -85,B 0,C 180,E1 -6923.288,E2 -6923.288} C_VEL
LIN {X 0,Y 480.93,Z 548.793,A -85,B 0,C 180,E1 -6924.55,E2 -6924.55} C_VEL
LIN {X 0,Y 480.827,Z 552.403,A -85,B 0,C 180,E1 -6925.81,E2 -6925.81} C_VEL
LIN {X 0,Y 480.888,Z 554.268,A -85,B 0,C 180,E1 -6926.649,E2 -6926.649} C_VEL
LIN {X 0,Y 480.792,Z 556.658,A -85,B 0,C 180,E1 -6928.325,E2 -6928.325} C_VEL
LIN {X 0,Y 480.76,Z 557.264,A -85,B 0,C 180,E1 -6929.163,E2 -6929.163} C_VEL
LIN {X 0,Y 480.743,Z 557.479,A -85,B 0,C 180,E1 -6930.001,E2 -6930.001} C_VEL
LIN {X 0,Y 480.792,Z 556.654,A -85,B 0,C 180,E1 -6931.676,E2 -6931.676} C_VEL
LIN {X 0,Y 480.888,Z 554.26,A -85,B 0,C 180,E1 -6933.352,E2 -6933.352} C_VEL
LIN {X 0,Y 480.839,Z 551.318,A -85,B 0,C 180,E1 -6934.611,E2 -6934.611} C_VEL
LIN {X 0,Y 480.928,Z 547.343,A -85,B 0,C 180,E1 -6935.872,E2 -6935.872} C_VEL
LIN {X 0,Y 481.109,Z 541.233,A -85,B 0,C 180,E1 -6937.344,E2 -6937.344} C_VEL
LIN {X 0,Y 481.319,Z 534.557,A -85,B 0,C 180,E1 -6938.608,E2 -6938.608} C_VEL
LIN {X 0,Y 481.657,Z 526.279,A -85,B 0,C 180,E1 -6939.873,E2 -6939.873} C_VEL
LIN {X 0,Y 482.012,Z 517.799,A -85,B 0,C 180,E1 -6940.927,E2 -6940.927} C_VEL
LIN {X 0,Y 482.485,Z 507.351,A -85,B 0,C 180,E1 -6941.979,E2 -6941.979} C_VEL
LIN {X 0,Y 482.872,Z 496.064,A -85,B 0,C 180,E1 -6942.894,E2 -6942.894} C_VEL
LIN {X 0,Y 483.378,Z 483.762,A -85,B 0,C 180,E1 -6943.667,E2 -6943.667} C_VEL
LIN {X 0,Y 483.844,Z 471.497,A -85,B 0,C 180,E1 -6944.243,E2 -6944.243} C_VEL
LIN {X 0,Y 484.184,Z 458.966,A -85,B 0,C 180,E1 -6944.662,E2 -6944.662} C_VEL
LIN {X 0,Y 484.35,Z 446.172,A -85,B 0,C 180,E1 -6944.926,E2 -6944.926} C_VEL
LIN {X 0,Y 484.802,Z 360.568,A -85,B 0,C 180,E1 -6946.21,E2 -6946.21} C_VEL
LIN {X 0,Y 482.295,Z 344.715,A -85,B 0,C 180,E1 -6946.564,E2 -6946.564} C_VEL
LIN {X 0,Y 482.815,Z 329.638,A -85,B 0,C 180,E1 -6949.148,E2 -6949.148} C_VEL
LIN {X 0,Y 483.46,Z 313.276,A -85,B 0,C 180,E1 -6951.991,E2 -6951.991} C_VEL
LIN {X 0,Y 483.64,Z 305.866,A -85,B 0,C 180,E1 -6953.301,E2 -6953.301} C_VEL
LIN {X 0,Y 481.648,Z 295.492,A -85,B 0,C 180,E1 -6955.288,E2 -6955.288} C_VEL
LIN {X 0,Y 481.694,Z 295.49,A -85,B 0,C 180,E1 -6957.833,E2 -6957.833} C_VEL
LIN {X 0,Y 481.647,Z 295.491,A -85,B 0,C 180,E1 -6960.711,E2 -6960.711} C_VEL
LIN {X 0,Y 481.7,Z 295.487,A -85,B 0,C 180,E1 -6963.733,E2 -6963.733} C_VEL
LIN {X 0,Y 481.622,Z 295.49,A -85,B 0,C 180,E1 -6966.748,E2 -6966.748} C_VEL
LIN {X 0,Y 481.66,Z 295.488,A -85,B 0,C 180,E1 -6969.942,E2 -6969.942} C_VEL
LIN {X 0,Y 481.628,Z 295.487,A -85,B 0,C 180,E1 -6973.146,E2 -6973.146} C_VEL
LIN {X 0,Y 481.654,Z 295.484,A -85,B 0,C 180,E1 -6975.642,E2 -6975.642} C_VEL
LIN {X 0,Y 481.65,Z 295.487,A -85,B 0,C 180,E1 -6978.958,E2 -6978.958} C_VEL
LIN {X 0,Y 481.651,Z 295.482,A -85,B 0,C 180,E1 -6981.994,E2 -6981.994} C_VEL
LIN {X 0,Y 481.689,Z 295.48,A -85,B 0,C 180,E1 -6985.318,E2 -6985.318} C_VEL
LIN {X 0,Y 481.645,Z 295.483,A -85,B 0,C 180,E1 -6988.312,E2 -6988.312} C_VEL
LIN {X 0,Y 481.676,Z 295.484,A -85,B 0,C 180,E1 -6991.217,E2 -6991.217} C_VEL
LIN {X 0,Y 481.664,Z 295.482,A -85,B 0,C 180,E1 -6994.041,E2 -6994.041} C_VEL
LIN {X 0,Y 481.675,Z 295.483,A -85,B 0,C 180,E1 -6996.812,E2 -6996.812} C_VEL
LIN {X 0,Y 481.696,Z 295.483,A -85,B 0,C 180,E1 -6999.503,E2 -6999.503} C_VEL
LIN {X 0,Y 481.692,Z 295.477,A -85,B 0,C 180,E1 -7002.158,E2 -7002.158} C_VEL
LIN {X 0,Y 481.743,Z 295.471,A -85,B 0,C 180,E1 -7004.776,E2 -7004.776} C_VEL
LIN {X 0,Y 481.751,Z 295.47,A -85,B 0,C 180,E1 -7008.215,E2 -7008.215} C_VEL
LIN {X 0,Y 481.739,Z 295.476,A -85,B 0,C 180,E1 -7011.611,E2 -7011.611} C_VEL
LIN {X 0,Y 481.805,Z 295.467,A -85,B 0,C 180,E1 -7014.14,E2 -7014.14} C_VEL
LIN {X 0,Y 481.918,Z 295.449,A -85,B 0,C 180,E1 -7017.493,E2 -7017.493} C_VEL
LIN {X 0,Y 481.94,Z 295.451,A -85,B 0,C 180,E1 -7020,E2 -7020} C_VEL
LIN {X 0,Y 481.92,Z 295.453,A -85,B 0,C 180,E1 -7022.508,E2 -7022.508} C_VEL
LIN {X 0,Y 481.798,Z 295.464,A -85,B 0,C 180,E1 -7025.861,E2 -7025.861} C_VEL
LIN {X 0,Y 481.741,Z 295.477,A -85,B 0,C 180,E1 -7028.389,E2 -7028.389} C_VEL
LIN {X 0,Y 481.752,Z 295.471,A -85,B 0,C 180,E1 -7031.785,E2 -7031.785} C_VEL
LIN {X 0,Y 481.744,Z 295.474,A -85,B 0,C 180,E1 -7035.224,E2 -7035.224} C_VEL
LIN {X 0,Y 481.71,Z 295.481,A -85,B 0,C 180,E1 -7038.722,E2 -7038.722} C_VEL
LIN {X 0,Y 481.647,Z 295.484,A -85,B 0,C 180,E1 -7041.395,E2 -7041.395} C_VEL
LIN {X 0,Y 481.658,Z 295.482,A -85,B 0,C 180,E1 -7044.114,E2 -7044.114} C_VEL
LIN {X 0,Y 481.697,Z 295.485,A -85,B 0,C 180,E1 -7047.127,E2 -7047.127} C_VEL
LIN {X 0,Y 481.674,Z 295.482,A -85,B 0,C 180,E1 -7049.742,E2 -7049.742} C_VEL
LIN {X 0,Y 481.672,Z 295.481,A -85,B 0,C 180,E1 -7052.675,E2 -7052.675} C_VEL
LIN {X 0,Y 481.634,Z 295.491,A -85,B 0,C 180,E1 -7055.71,E2 -7055.71} C_VEL
LIN {X 0,Y 481.673,Z 295.482,A -85,B 0,C 180,E1 -7058.859,E2 -7058.859} C_VEL
LIN {X 0,Y 481.649,Z 295.49,A -85,B 0,C 180,E1 -7061.912,E2 -7061.912} C_VEL
LIN {X 0,Y 481.657,Z 295.485,A -85,B 0,C 180,E1 -7064.458,E2 -7064.458} C_VEL
LIN {X 0,Y 481.632,Z 295.494,A -85,B 0,C 180,E1 -7067.837,E2 -7067.837} C_VEL
LIN {X 0,Y 481.669,Z 295.485,A -85,B 0,C 180,E1 -7071.14,E2 -7071.14} C_VEL
LIN {X 0,Y 481.661,Z 295.487,A -85,B 0,C 180,E1 -7074.797,E2 -7074.797} C_VEL
LIN {X 0,Y 481.722,Z 295.565,A -85,B 0,C 180,E1 -7077.843,E2 -7077.843} C_VEL
LIN {X 0,Y 482.618,Z 300.485,A -85,B 0,C 180,E1 -7078.845,E2 -7078.845} C_VEL
LIN {X 0,Y 482.563,Z 311.218,A -85,B 0,C 180,E1 -7080.908,E2 -7080.908} C_VEL
LIN {X 0,Y 482.393,Z 319.821,A -85,B 0,C 180,E1 -7082.513,E2 -7082.513} C_VEL
LIN {X 0,Y 485.041,Z 333.638,A -85,B 0,C 180,E1 -7082.824,E2 -7082.824} C_VEL
LIN {X 0,Y 484.961,Z 348.13,A -85,B 0,C 180,E1 -7083.042,E2 -7083.042} C_VEL
LIN {X 0,Y 484.21,Z 353.976,A -85,B 0,C 180,E1 -7083.104,E2 -7083.104} C_VEL
LIN {X 0,Y 478.581,Z 372.986,A -85,B 0,C 180,E1 -7083.188,E2 -7083.188} C_VEL
LIN {X 0,Y 477.897,Z 378.829,A -85,B 0,C 180,E1 -7083.253,E2 -7083.253} C_VEL
LIN {X 0,Y 477.526,Z 427.686,A -85,B 0,C 180,E1 -7084.019,E2 -7084.019} C_VEL
LIN {X 0,Y 477.222,Z 440.35,A -85,B 0,C 180,E1 -7084.378,E2 -7084.378} C_VEL
LIN {X 0,Y 476.87,Z 453.38,A -85,B 0,C 180,E1 -7084.931,E2 -7084.931} C_VEL
LIN {X 0,Y 476.468,Z 465.033,A -85,B 0,C 180,E1 -7085.606,E2 -7085.606} C_VEL
LIN {X 0,Y 475.97,Z 477.015,A -85,B 0,C 180,E1 -7086.504,E2 -7086.504} C_VEL
LIN {X 0,Y 475.408,Z 487.673,A -85,B 0,C 180,E1 -7087.51,E2 -7087.51} C_VEL
LIN {X 0,Y 475.005,Z 496.917,A -85,B 0,C 180,E1 -7088.601,E2 -7088.601} C_VEL
LIN {X 0,Y 474.589,Z 505.598,A -85,B 0,C 180,E1 -7089.861,E2 -7089.861} C_VEL
LIN {X 0,Y 474.313,Z 511.854,A -85,B 0,C 180,E1 -7090.975,E2 -7090.975} C_VEL
LIN {X 0,Y 474.066,Z 517.936,A -85,B 0,C 180,E1 -7092.307,E2 -7092.307} C_VEL
LIN {X 0,Y 473.912,Z 522.673,A -85,B 0,C 180,E1 -7093.634,E2 -7093.634} C_VEL
LIN {X 0,Y 473.871,Z 525.314,A -85,B 0,C 180,E1 -7094.585,E2 -7094.585} C_VEL
LIN {X 0,Y 473.683,Z 528.717,A -85,B 0,C 180,E1 -7096.267,E2 -7096.267} C_VEL
LIN {X 0,Y 473.68,Z 529.812,A -85,B 0,C 180,E1 -7097.14,E2 -7097.14} C_VEL
LIN {X 0,Y 473.746,Z 530.633,A -85,B 0,C 180,E1 -7098.27,E2 -7098.27} C_VEL
LIN {X 0,Y 473.665,Z 530.658,A -85,B 0,C 180,E1 -7099.743,E2 -7099.743} C_VEL
LIN {X 0,Y 473.719,Z 529.145,A -85,B 0,C 180,E1 -7101.468,E2 -7101.468} C_VEL
LIN {X 0,Y 473.75,Z 527.799,A -85,B 0,C 180,E1 -7102.327,E2 -7102.327} C_VEL
LIN {X 0,Y 473.855,Z 525.044,A -85,B 0,C 180,E1 -7103.576,E2 -7103.576} C_VEL
LIN {X 0,Y 473.921,Z 521.094,A -85,B 0,C 180,E1 -7104.895,E2 -7104.895} C_VEL
LIN {X 0,Y 474.139,Z 516.107,A -85,B 0,C 180,E1 -7106.175,E2 -7106.175} C_VEL
LIN {X 0,Y 474.297,Z 509.876,A -85,B 0,C 180,E1 -7107.452,E2 -7107.452} C_VEL
LIN {X 0,Y 474.733,Z 502.059,A -85,B 0,C 180,E1 -7108.727,E2 -7108.727} C_VEL
LIN {X 0,Y 475.109,Z 492.374,A -85,B 0,C 180,E1 -7109.999,E2 -7109.999} C_VEL
LIN {X 0,Y 475.485,Z 483.43,A -85,B 0,C 180,E1 -7110.952,E2 -7110.952} C_VEL
LIN {X 0,Y 476.045,Z 472.333,A -85,B 0,C 180,E1 -7111.903,E2 -7111.903} C_VEL
LIN {X 0,Y 476.468,Z 461.515,A -85,B 0,C 180,E1 -7112.641,E2 -7112.641} C_VEL
LIN {X 0,Y 476.818,Z 449.604,A -85,B 0,C 180,E1 -7113.274,E2 -7113.274} C_VEL
LIN {X 0,Y 477.12,Z 437.371,A -85,B 0,C 180,E1 -7113.747,E2 -7113.747} C_VEL
LIN {X 0,Y 477.35,Z 424.761,A -85,B 0,C 180,E1 -7114.062,E2 -7114.062} C_VEL
LIN {X 0,Y 478.046,Z 334.541,A -85,B 0,C 180,E1 -7115.43,E2 -7115.43} C_VEL
LIN {X 0,Y 475.265,Z 319.88,A -85,B 0,C 180,E1 -7115.754,E2 -7115.754} C_VEL
LIN {X 0,Y 475.88,Z 304.804,A -85,B 0,C 180,E1 -7118.706,E2 -7118.706} C_VEL
LIN {X 0,Y 475.052,Z 298.453,A -85,B 0,C 180,E1 -7120.01,E2 -7120.01} C_VEL
LIN {X 0,Y 474.679,Z 296.358,A -85,B 0,C 180,E1 -7120.449,E2 -7120.449} C_VEL
LIN {X 0,Y 474.645,Z 296.361,A -85,B 0,C 180,E1 -7122.832,E2 -7122.832} C_VEL
LIN {X 0,Y 474.654,Z 296.36,A -85,B 0,C 180,E1 -7125.754,E2 -7125.754} C_VEL
LIN {X 0,Y 474.66,Z 296.354,A -85,B 0,C 180,E1 -7129.01,E2 -7129.01} C_VEL
LIN {X 0,Y 474.589,Z 296.366,A -85,B 0,C 180,E1 -7131.728,E2 -7131.728} C_VEL
LIN {X 0,Y 474.626,Z 296.363,A -85,B 0,C 180,E1 -7134.494,E2 -7134.494} C_VEL
LIN {X 0,Y 474.597,Z 296.362,A -85,B 0,C 180,E1 -7137.325,E2 -7137.325} C_VEL
LIN {X 0,Y 474.586,Z 296.369,A -85,B 0,C 180,E1 -7140.23,E2 -7140.23} C_VEL
LIN {X 0,Y 474.613,Z 296.36,A -85,B 0,C 180,E1 -7143.221,E2 -7143.221} C_VEL
LIN {X 0,Y 474.576,Z 296.369,A -85,B 0,C 180,E1 -7146.323,E2 -7146.323} C_VEL
LIN {X 0,Y 474.597,Z 296.362,A -85,B 0,C 180,E1 -7149.642,E2 -7149.642} C_VEL
LIN {X 0,Y 474.571,Z 296.366,A -85,B 0,C 180,E1 -7152.229,E2 -7152.229} C_VEL
LIN {X 0,Y 474.608,Z 296.364,A -85,B 0,C 180,E1 -7155.297,E2 -7155.297} C_VEL
LIN {X 0,Y 474.586,Z 296.363,A -85,B 0,C 180,E1 -7158.21,E2 -7158.21} C_VEL
LIN {X 0,Y 474.592,Z 296.365,A -85,B 0,C 180,E1 -7161.54,E2 -7161.54} C_VEL
LIN {X 0,Y 474.604,Z 296.363,A -85,B 0,C 180,E1 -7164.723,E2 -7164.723} C_VEL
LIN {X 0,Y 474.602,Z 296.363,A -85,B 0,C 180,E1 -7167.785,E2 -7167.785} C_VEL
LIN {X 0,Y 474.569,Z 296.367,A -85,B 0,C 180,E1 -7170.894,E2 -7170.894} C_VEL
LIN {X 0,Y 474.563,Z 296.373,A -85,B 0,C 180,E1 -7173.622,E2 -7173.622} C_VEL
LIN {X 0,Y 474.626,Z 296.358,A -85,B 0,C 180,E1 -7176.641,E2 -7176.641} C_VEL
LIN {X 0,Y 474.637,Z 296.36,A -85,B 0,C 180,E1 -7180.088,E2 -7180.088} C_VEL
LIN {X 0,Y 474.575,Z 296.364,A -85,B 0,C 180,E1 -7182.771,E2 -7182.771} C_VEL
LIN {X 0,Y 474.593,Z 296.365,A -85,B 0,C 180,E1 -7185.419,E2 -7185.419} C_VEL
LIN {X 0,Y 474.683,Z 296.359,A -85,B 0,C 180,E1 -7188.037,E2 -7188.037} C_VEL
LIN {X 0,Y 474.654,Z 296.356,A -85,B 0,C 180,E1 -7191.485,E2 -7191.485} C_VEL
LIN {X 0,Y 474.725,Z 296.353,A -85,B 0,C 180,E1 -7194.052,E2 -7194.052} C_VEL
LIN {X 0,Y 474.87,Z 296.328,A -85,B 0,C 180,E1 -7197.455,E2 -7197.455} C_VEL
LIN {X 0,Y 474.867,Z 296.332,A -85,B 0,C 180,E1 -7200,E2 -7200} C_VEL
LIN {X 0,Y 474.867,Z 296.335,A -85,B 0,C 180,E1 -7202.545,E2 -7202.545} C_VEL
LIN {X 0,Y 474.747,Z 296.344,A -85,B 0,C 180,E1 -7205.948,E2 -7205.948} C_VEL
LIN {X 0,Y 474.691,Z 296.358,A -85,B 0,C 180,E1 -7208.514,E2 -7208.514} C_VEL
LIN {X 0,Y 474.694,Z 296.35,A -85,B 0,C 180,E1 -7211.963,E2 -7211.963} C_VEL
LIN {X 0,Y 474.671,Z 296.352,A -85,B 0,C 180,E1 -7215.767,E2 -7215.767} C_VEL
LIN {X 0,Y 474.652,Z 296.363,A -85,B 0,C 180,E1 -7219.011,E2 -7219.011} C_VEL
LIN {X 0,Y 474.578,Z 296.365,A -85,B 0,C 180,E1 -7221.729,E2 -7221.729} C_VEL
LIN {X 0,Y 474.618,Z 296.36,A -85,B 0,C 180,E1 -7224.495,E2 -7224.495} C_VEL
LIN {X 0,Y 474.665,Z 296.36,A -85,B 0,C 180,E1 -7227.333,E2 -7227.333} C_VEL
LIN {X 0,Y 474.596,Z 296.362,A -85,B 0,C 180,E1 -7230.231,E2 -7230.231} C_VEL
LIN {X 0,Y 474.627,Z 296.364,A -85,B 0,C 180,E1 -7233.221,E2 -7233.221} C_VEL
LIN {X 0,Y 474.577,Z 296.364,A -85,B 0,C 180,E1 -7236.325,E2 -7236.325} C_VEL
LIN {X 0,Y 474.619,Z 296.367,A -85,B 0,C 180,E1 -7239.548,E2 -7239.548} C_VEL
LIN {X 0,Y 474.594,Z 296.364,A -85,B 0,C 180,E1 -7242.234,E2 -7242.234} C_VEL
LIN {X 0,Y 474.611,Z 296.362,A -85,B 0,C 180,E1 -7245.299,E2 -7245.299} C_VEL
LIN {X 0,Y 474.61,Z 296.364,A -85,B 0,C 180,E1 -7248.215,E2 -7248.215} C_VEL
LIN {X 0,Y 474.605,Z 296.363,A -85,B 0,C 180,E1 -7251.543,E2 -7251.543} C_VEL
LIN {X 0,Y 474.618,Z 296.36,A -85,B 0,C 180,E1 -7254.726,E2 -7254.726} C_VEL
LIN {X 0,Y 474.633,Z 296.361,A -85,B 0,C 180,E1 -7257.789,E2 -7257.789} C_VEL
LIN {X 0,Y 474.619,Z 296.361,A -85,B 0,C 180,E1 -7260.886,E2 -7260.886} C_VEL
LIN {X 0,Y 474.625,Z 296.362,A -85,B 0,C 180,E1 -7263.627,E2 -7263.627} C_VEL
LIN {X 0,Y 474.662,Z 296.501,A -85,B 0,C 180,E1 -7264.713,E2 -7264.713} C_VEL
LIN {X 0,Y 476.652,Z 307.449,A -85,B 0,C 180,E1 -7266.771,E2 -7266.771} C_VEL
LIN {X 0,Y 475.956,Z 325.398,A -85,B 0,C 180,E1 -7269.922,E2 -7269.922} C_VEL
LIN {X 0,Y 475.402,Z 340.729,A -85,B 0,C 180,E1 -7272.582,E2 -7272.582} C_VEL
LIN {X 0,Y 475.271,Z 344.735,A -85,B 0,C 180,E1 -7273.273,E2 -7273.273} C_VEL
LIN {X 0,Y 477.988,Z 363.536,A -85,B 0,C 180,E1 -7273.658,E2 -7273.658} C_VEL
LIN {X 0,Y 477.389,Z 452.636,A -85,B 0,C 180,E1 -7275.017,E2 -7275.017} C_VEL
LIN {X 0,Y 476.965,Z 466.029,A -85,B 0,C 180,E1 -7275.385,E2 -7275.385} C_VEL
LIN {X 0,Y 476.593,Z 478.837,A -85,B 0,C 180,E1 -7275.919,E2 -7275.919} C_VEL
LIN {X 0,Y 476.202,Z 490.21,A -85,B 0,C 180,E1 -7276.56,E2 -7276.56} C_VEL
LIN {X 0,Y 475.677,Z 501.178,A -85,B 0,C 180,E1 -7277.352,E2 -7277.352} C_VEL
LIN {X 0,Y 475.208,Z 512.439,A -85,B 0,C 180,E1 -7278.376,E2 -7278.376} C_VEL
LIN {X 0,Y 474.781,Z 521.036,A -85,B 0,C 180,E1 -7279.338,E2 -7279.338} C_VEL
LIN {X 0,Y 474.474,Z 528.965,A -85,B 0,C 180,E1 -7280.408,E2 -7280.408} C_VEL
LIN {X 0,Y 474.162,Z 536.707,A -85,B 0,C 180,E1 -7281.692,E2 -7281.692} C_VEL
LIN {X 0,Y 473.935,Z 543.831,A -85,B 0,C 180,E1 -7283.188,E2 -7283.188} C_VEL
LIN {X 0,Y 473.844,Z 548.571,A -85,B 0,C 180,E1 -7284.468,E2 -7284.468} C_VEL
LIN {X 0,Y 473.734,Z 552.189,A -85,B 0,C 180,E1 -7285.747,E2 -7285.747} C_VEL
LIN {X 0,Y 473.795,Z 554.059,A -85,B 0,C 180,E1 -7286.599,E2 -7286.599} C_VEL
LIN {X 0,Y 473.741,Z 555.458,A -85,B 0,C 180,E1 -7287.45,E2 -7287.45} C_VEL
LIN {X 0,Y 473.688,Z 557.064,A -85,B 0,C 180,E1 -7289.151,E2 -7289.151} C_VEL
LIN {X 0,Y 473.67,Z 557.281,A -85,B 0,C 180,E1 -7290.001,E2 -7290.001} C_VEL
LIN {X 0,Y 473.688,Z 557.067,A -85,B 0,C 180,E1 -7290.851,E2 -7290.851} C_VEL
LIN {X 0,Y 473.741,Z 555.465,A -85,B 0,C 180,E1 -7292.551,E2 -7292.551} C_VEL
LIN {X 0,Y 473.795,Z 554.072,A -85,B 0,C 180,E1 -7293.402,E2 -7293.402} C_VEL
LIN {X 0,Y 473.762,Z 551.136,A -85,B 0,C 180,E1 -7294.681,E2 -7294.681} C_VEL
LIN {X 0,Y 473.835,Z 547.167,A -85,B 0,C 180,E1 -7295.96,E2 -7295.96} C_VEL
LIN {X 0,Y 474.02,Z 541.071,A -85,B 0,C 180,E1 -7297.455,E2 -7297.455} C_VEL
LIN {X 0,Y 474.281,Z 534.409,A -85,B 0,C 180,E1 -7298.737,E2 -7298.737} C_VEL
LIN {X 0,Y 474.607,Z 526.146,A -85,B 0,C 180,E1 -7300.021,E2 -7300.021} C_VEL
LIN {X 0,Y 475.035,Z 517.695,A -85,B 0,C 180,E1 -7301.089,E2 -7301.089} C_VEL
LIN {X 0,Y 475.512,Z 507.474,A -85,B 0,C 180,E1 -7302.14,E2 -7302.14} C_VEL
LIN {X 0,Y 475.959,Z 495.681,A -85,B 0,C 180,E1 -7303.111,E2 -7303.111} C_VEL
LIN {X 0,Y 476.481,Z 483.81,A -85,B 0,C 180,E1 -7303.868,E2 -7303.868} C_VEL
LIN {X 0,Y 476.97,Z 471.634,A -85,B 0,C 180,E1 -7304.452,E2 -7304.452} C_VEL
LIN {X 0,Y 477.343,Z 459.253,A -85,B 0,C 180,E1 -7304.877,E2 -7304.877} C_VEL
LIN {X 0,Y 477.511,Z 446.939,A -85,B 0,C 180,E1 -7305.144,E2 -7305.144} C_VEL
LIN {X 0,Y 478.038,Z 361.46,A -85,B 0,C 180,E1 -7306.446,E2 -7306.446} C_VEL
LIN {X 0,Y 475.323,Z 344.614,A -85,B 0,C 180,E1 -7306.814,E2 -7306.814} C_VEL
